	tonLimitPosMinReachedDelay	: TON;					// Timer osoiągniecia minimalnej wyskości 
	tonLimitPosMaxReachedDelay	: TON;					// Timer osiągnięcia maksymalnej wyskości
	tonSortingEngineOn			: TON;					// Opóźnienie po załączeniu napędu
	tonSortingEngineOff			: TON;					// Opóźnienie wyłączenia napędu
	tonSleeveFullEngineOn		: TON;					// Czas załączenia napędu po wykrciu braku nasadek
	tonEngineBlocked			: TON;					// Zablokowany silnik	
	rtCapSorterSensor			: R_TRIG;				// Triger
	tonTryUnblockWheel			: TON;					// Czas ruchu falownika w drugą stronę
	tofCapFeederSorterCapSensor	: TOF;					// Opóźnienie sygnału z czujnika obecności nasadki ultradzwiek
	tonCapFeederSorterCapSensor	: TON;					// Opóźnienie sygnału z czujnika obecności nasadki ultradźwięk
	tonAirBeforeStart			: TON;					// Czasówka opóźeniani przedmuchu
	tonAirBeforeStart2			: TON;					// Czasówka opóźeniani przedmuchu
	tonAirAfterStop				: TON;					// Czasówka przedmuchu po zatrzymaniu
	tonStoppingTime				: TON;					// Czasówka zbyt długiego zatrzymawania

	
	tonErrorHeightChange		: TON; 					// Timer błędu zacięcia się podnośnika
	tonMaxHeightError			: TON;					// Timer ustawienia zbyt dużej wysokości stacji
	tonMinHeightError			: TON;					// Timer ustawienia zbyt małej wysokości stacji
	tonCycleTimer				: TON;					// Czasówka cyklu
	rtrigCycleTimerRead			: R_TRIG;				// Trigger do statystyk cyklu 
	
	rtResetCommands				: R_TRIG;
	tonHomingSensor: TON;
	TimerOn: TON;
	TimerOff: TON;
	bImpOn: BOOL;
	rtCapFeederSorterCapSensor: R_TRIG;
	bBlowDelay: BOOL;
	tonbBlowDelay: TON;
	
	fbInverter: FB_MitsubishiInverter;
	fbInverter2: FB_MitsubishiInverter;	
	tonInverterError: TON;
	tonInverter2Error: TON;	
	tonbCapping1Tool2ActuatorUpError: TON;
	tonbCapping2Tool2ActuatorUpError: TON;	
	
	(*Ostrzeżenia*)
	fbbLevelSensor:	FB_InputFilter;
	(*Inne*)	

	tonGates1	:	TON;	//Czasówka dla szlabanów w rękawe
	tonGates2	:	TON;	//Czasówka dla szlabanów w rękawe
	tonGates3	:	TON;	//Czasówka dla szlabanów w rękawe
	tonGates4	:	TON;	//Czasówka dla szlabanów w rękawe

	toneHolding1 :TON;
	toneHolding2 :TON;
	toneGoingUp	:TON;
	toneHolding1Tool2 :TON;
	toneHolding2Tool2 :TON;
	
	bDone1				: BOOL;					// Sygnał o niezakończonym cyklu
	bDone2				: BOOL;					// Sygnał o niezakończonym cyklu
	
	tonDown1:TON;
	tonDown2:TON;	
	tonEnginesRun:TON;	
	tonDone	:TON;	
	ftbRunEngine: F_TRIG;
	bGates	    :	BOOL;	//Controla szłabanow w rękawe  
	bTryUnblockWheel : BOOL;
	iTryUnblockWheel : INT;
END_VAR

//Wywołanie bloczków od stacji. Ważna jest ich kolejność!!!
ACT_Limits();
ACT_HeightMotor();
ACT_ErrorHandling();

ACT_Signals();
ACT_Control();
aEngine();
ACT_Inverter();
ACT_Statistic();
ACT_Status();
ACT_Warnings();
aStationID();	

lrLastHeightMotorPositionCV:=lrHeightMotorCV;

ACTION ACT_Control:
	(*****Wyłączenie enable*****)
	IF NOT bEnable THEN
		IF eState <> E_Station.eDisabled AND eState <> E_Station.ePreparingToDisable THEN
				eState 				:= E_Station.ePreparingToDisable; 
		END_IF	
	END_IF

	(*****Estop*****)
	IF NOT bEstop  THEN	
		IF eState <> E_Station.eAborted AND eState <> E_Station.eAborting AND eState <> E_Station.eDisabled THEN
				eState 				:= E_Station.eAborting; 
		END_IF
	END_IF


	CASE eState OF
//--------------------------------------------------------------------------------
// Stan maszyny po wyłączeniu i przygotowanie do uruchomienia
	E_Station.eDisabled: 					// Stan nieaktywnosci (Stacja wyłączona) 
	
		IF bEnable THEN
			eState 				:= E_Station.ePreparingToReady; 
		END_IF 
		
//--------------------------------------------------------------------------------
// Stan maszyny po zatrzymaniu awaryjnym   
	E_Station.eAborted: 					// Stan bezpiecznego zatrzymania (po Abortingu) 

		IF bEStop THEN
			eState 				:= E_Station.ePreparingToReady;
		END_IF
		
//--------------------------------------------------------------------------------
// Stan maszyny naciśnieciu estopa 	
	E_Station.eAborting:                 	// Stan bezpiecznego zatrzymywania (po EStopie)

		ACT_ResetCommands();

		eState 						:=  E_Station.eAborted;  
		eRunningState				:=	E_GripperScrewer.eReady;
		
//--------------------------------------------------------------------------------
// Stan masyzny po wykryciu błędu			
	E_Station.eError:                 	 	// Stan błędu 	
		
		ACT_ResetCommands();
		
		IF bReset THEN
			eState 					:= E_Station.eResetting;
			bError					 := FALSE;
		END_IF
		
//--------------------------------------------------------------------------------
// Stan masyzny po wykryciu błędu
	E_Station.eResetting:					// Stan resetowania bledu (po Errorze)
			CASE udiErrorID OF
		
				//Error - Błąd falownika
				353,354:
					fbInverter.bReset	:= TRUE;
					fbInverter2.bReset	:= TRUE;					
					bError 				:= FALSE;
				ELSE
					bError := FALSE;	
			END_CASE		
		
		IF NOT bError AND fbInverter.eState = E_Station.eReady THEN
			fbInverter.bReset	:= FALSE;	
			fbInverter2.bReset	:= FALSE;
			//{warning 'Sprawdzić błąd falownika CapFeeder'}
			udiErrorID 			:=	0;
			sErrorDescription 	:=	'';
			eState 				:=	E_Station.ePreparingToReady;
			eRunningState		:=	E_GripperScrewer.eReady;
		ELSE
			eState 				:=	E_Station.eError;
		END_IF
    
//--------------------------------------------------------------------------------
// Stan ruchoow manualnych
	E_Station.eManualMovement:     			// Stan ruchów manualnych  
   
		ACT_ManualMovements();
		//Wyjście z trybu serwisowego
		IF NOT bManualMovement THEN
			bHeightMotorUp				:=	FALSE;
			bHeightMotorDown			:=	FALSE;
			eState:=E_Station.eReady;
		END_IF
		
//--------------------------------------------------------------------------------
// Stan rozpoczecia bazowania
	E_Station.eHoming:						// Stan bazowania 
		
		ACT_Homing();
		IF NOT bHoming AND NOT bHeightSet THEN
			bHeightMotorDown				:=	FALSE;
			bHeightMotorUp					:=	FALSE;
		   eState							:=	E_Station.ePreparingToReady;
		END_IF		
		
//--------------------------------------------------------------------------------
// Stan zakończenia bazowania
	E_Station.eHomingDone:                  // Stan wykonania bazowania 
	
		bHeightMotorDown					:=	FALSE;
		bHeightMotorUp						:=	FALSE;
		bHeightMotorEncoderCounterReset		:=	FALSE;
		bHomingDone							:=	TRUE;
		IF NOT bHoming AND NOT bHeightSet THEN
		   eState:=E_Station.eReady;
		END_IF
		
//--------------------------------------------------------------------------------
// Stan przygotowania do gotowości
	E_Station.ePreparingToReady:            // Stan przygotowywania do gotowosci (zawsze przed Ready)  

		eRunningState	:=	E_GripperScrewer.eReady;
		eState			:=	E_Station.eReady;	
		
//-------------------------------------------------------------------------------
// Stan przygotowania do wyłączenia maszyny
	E_Station.ePreparingToDisable:          // Stan przygotowywania do nieaktywnosci (po wyłączeniu Enable) 

		bHeightMotorUp		:=	TRUE;
		bHeightMotorDown	:=	FALSE;	
		IF tonHeightNoChange.Q OR tonHeightNoChangeTime.Q THEN
			bHeightMotorUp			:=	FALSE;
			bHeightMotorDown		:=	FALSE;	
			eRunningState			:=	E_GripperScrewer.eReady;		
			eState					:=	E_Station.eDisabled;
		END_IF	
			
//--------------------------------------------------------------------------------
// Stan gotowości
	E_Station.eReady:						// Stan gotowosci 
	
		(*Skasowanie wszystkich komend*)
		IF rtResetCommands.Q THEN	ACT_ResetCommands();	END_IF
	
		IF (bRun1 OR bRun2) AND NOT bCycleDone1 AND NOT bCycleNotDone1 AND NOT bCycleDone2 AND NOT bCycleNotDone2 THEN
			eState 				:= E_Station.eStarting; 
		END_IF
		IF bHoming OR bHeightSet THEN
			eState 				:= E_Station.eHoming; 
		END_IF
		IF bManualMovement THEN
			bManualHeightMotorUp					:=	bHeightMotorUp;					
			bManualHeightMotorDown				:=	bHeightMotorDown;	
			bManualEngine1						:=	fbInverter.bRun;							
			bManualEngine2						:=	fbInverter2.bRun;		
			bManualCapping1Tool1Actuator		:=	bCapping1Tool1Actuator;		
			bManualCapping2Tool1Actuator		:=	bCapping2Tool1Actuator;		
			bManualCapping12Tool1BlockActuator	:=	bCapping12Tool1BlockActuator;
			bManualCappingBlockActuator			:=	bCappingBlockActuator;	
			bManualCapping1Tool2Down			:=	bCapping1Tool2Down;	
			bManualCapping1Tool2Tight			:=	bCapping1Tool2Tight;			
			bManualCapping1Tool2Realese			:=	bCapping1Tool2Realese;		
			bManualCapping2Tool2Down			:=	bCapping2Tool2Down;				
			bManualCapping2Tool2Tight			:=	bCapping2Tool2Tight;
			bManualCapping2Tool2Realese			:=	bCapping2Tool2Realese;
			bManualFormPositioning				:=	bFormPositioning;			
			eState 								:=	E_Station.eManualMovement; 
		END_IF
		IF NOT bRun1 AND NOT bRun2 THEN
			bDone1						:= FALSE;
			bDone2						:= FALSE;
			bCycleDone1 				:= FALSE;
			bCycleNotDone1 				:= FALSE;	
			bCycleDone2					:= FALSE;
			bCycleNotDone2 				:= FALSE;	
			bWarning1					:= FALSE;	
		END_IF
		
//--------------------------------------------------------------------------------
// Stan zatrzymywania
	E_Station.eStopping:					// Stan zatrzymywania 
		
		ACT_Running();

		IF tonStoppingTime.Q THEN
			ACT_ResetCommands();
			eRunningState							:= E_GripperScrewer.eReady;
			eState									:= E_Station.eReady;
		END_IF

		
//--------------------------------------------------------------------------------
// Stan uruchomienia lini ( po eReady)
	E_Station.eStarting:                  	// Stan uruchamiania (po Ready)

		eState					 := E_Station.eRunning; 

//--------------------------------------------------------------------------------
// Stan wykonywania pracy
	E_Station.eRunning:               		// Stan wykonywania cyklu (po Startingu), w tym stanie osobny

		ACT_Running();
		IF NOT bRun1 AND NOT bRun2 THEN					(*Przerywanie cyklu*)
			eState 				 := E_Station.eStopping;	
		END_IF
		IF (bCycleDone1 OR bCycleNotDone1) AND (bCycleDone2 OR bCycleNotDone2)  THEN (*Cykl zakończony*)
			eState 				 := E_Station.eReady;
		END_IF						
		
		
END_CASE
END_ACTION

ACTION ACT_ErrorHandling:
//OBSŁUGA BŁĘDÓW STACJI SPRAWDZANIA
//************LISTA BŁĘDÓW***************
bStateError:= (eState=E_Station.eError) OR (eState=E_Station.eResetting) OR bIgnoreError;
//************LISTA BŁĘDÓW***************

//Error 1 - podnośnik nie porusza się pomimo wysterowania 
tonErrorHeightChange(IN:=(bHeightMotorUp OR bHeightMotorDown) AND lrLastHeightMotorPositionCV=lrHeightMotorCV, PT:=T#3S);
tonMaxHeightError	(IN:=lrHeightMotorSV>lrMaxHeight AND NOT bHomingNeeded AND eState=E_Station.eReady,PT:=T#30S);
tonMinHeightError	(IN:=lrHeightMotorSV<lrMinHeight AND NOT bHomingNeeded AND eState=E_Station.eReady,PT:=T#30S);
tonInverterError	(IN:=fbInverter.bError AND NOT bStateError, PT:=T#3S);
tonInverter2Error	(IN:=fbInverter2.bError AND NOT bStateError, PT:=T#3S);

tonbCapping1Tool2ActuatorUpError (IN:= iTool = 2 (*G.dociskająca*) AND NOT IbCapping1Tool2ActuatorUpSensor AND NOT bCapping1Tool2Down, PT:=T#2S);
tonbCapping2Tool2ActuatorUpError (IN:= iTool = 2 (*G.dociskająca*) AND NOT IbCapping2Tool2ActuatorUpSensor AND NOT bCapping2Tool2Down, PT:=T#2S);

IF (bEnable OR (eState = E_Station.ePreparingToDisable)) AND NOT bIgnoreError THEN
	
	IF tonErrorHeightChange.Q THEN
		bError:=TRUE;
		udiErrorID:=350;
		sErrorDescription:='Blokada podnośnika lub brak zasilania - sprawdź czujnik lub odblokuj mechanicznie';	
		sErrorDescription2:='';
	END_IF
	
	//Error - Bład nastaw max
	IF tonMaxHeightError.Q  THEN
		bError:=TRUE;
		udiErrorID:=351;
		sErrorDescription:='Wartość zadana wysokości jest większa od maksymalnej - zmień ustawienia w recepturze';
		sErrorDescription2:=REAL_TO_STRING(LREAL_TO_INT(lrMaxHeight));
	END_IF
	
	//Error - Bład nastaw min
	IF tonMinHeightError.Q THEN
		bError:=TRUE;
		udiErrorID:=352;
		sErrorDescription:='Wartość zadana wysokości jest mniejsza od minimalnej - zmień ustawienia w recepturze';
		sErrorDescription2:=REAL_TO_STRING(LREAL_TO_INT(lrMinHeight));
	END_IF	
	
	//Error - Bład falownika 1
	IF tonInverterError.Q THEN
		bError:=TRUE;
		udiErrorID:=353;
		sErrorDescription:='Błąd falownika głowicy 1';
		sErrorDescription2:='';
	END_IF		
	
	//Error - Bład falownika 2
	IF tonInverter2Error.Q THEN
		bError:=TRUE;
		udiErrorID:=354;
		sErrorDescription:='Błąd falownika głowicy 2';
		sErrorDescription2:='';
	END_IF			
	
	//Error Glowica 1 - Bład góry
	IF tonbCapping1Tool2ActuatorUpError.Q THEN
		bError:=TRUE;
		udiErrorID:=355;
		sErrorDescription:='Błąd górnej pozycji głowicy dociskającej 1- upewnij się że jest wybrane dobre narzędzie lub sprawdź czujnik';
		sErrorDescription2:='';	
	END_IF			
	//Error Glowica 2 - Bład góry
	IF tonbCapping2Tool2ActuatorUpError.Q THEN
		bError:=TRUE;
		udiErrorID:=356;
		sErrorDescription:='Błąd górnej pozycji głowicy dociskającej 2 - upewnij się że jest wybrane dobre narzędzie lub sprawdź czujnik';
		sErrorDescription2:='';	
	END_IF			
	
ELSE
	bError	:=FALSE;
END_IF


//-----------------------------------------------------------------------
IF bError AND NOT bStateError THEN

	IF eLastState = eRunning THEN
		bCycleNotDone1						:= TRUE;
	END_IF

	eState 									:= E_Station.eError;
END_IF


//------------------------------------------------------------------------

(*Wyświetlanie błedu na wyjściu*)
bError;

(*Przepisywanie nazwy stacji*)
sErrorStationName 							:= sStationName;

//Jezeli nie zbazowane to potrzebne bazowanie
IF NOT bHeightMotorEncoderHomed  THEN
	bHomingDone								:=	FALSE;
END_IF
END_ACTION

ACTION ACT_HeightMotor:
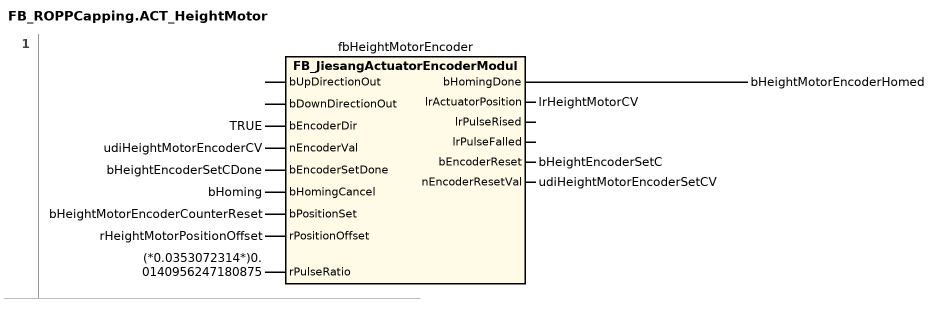
// NETWORK 1
fbHeightMotorEncoder(
    bEncoderDir := TRUE,
    nEncoderVal := udiHeightMotorEncoderCV,
    bEncoderSetDone := bHeightEncoderSetCDone,
    bHomingCancel := bHoming,
    bPositionSet := bHeightMotorEncoderCounterReset,
    rPositionOffset := rHeightMotorPositionOffset,
    rPulseRatio := (*0.0353072314*)0.0140956247180875,
    lrActuatorPosition => lrHeightMotorCV,
    bEncoderReset => bHeightEncoderSetC,
    nEncoderResetVal => udiHeightMotorEncoderSetCV); // FB_JiesangActuatorEncoderModul
bHeightMotorEncoderHomed := fbHeightMotorEncoder.bHomingDone;
END_ACTION

ACTION ACT_Homing:
//BAZOWANIE

tofHeightMotorDown(IN:=bHeightMotorDown, PT:=T#1S); //Zabezpieczenie przed zbyt szybkim przełączeniem pomiędzy Down a Up, bezpiecznieki sie palą
	
//Podnoszenie stacji do maksymalnej pozycji
IF NOT bHeightMotorEncoderHomed OR rtEncoderHomed.Q THEN
	bHeightMotorUp:=(*TRUE*) NOT tofHeightMotorDown.Q AND NOT tonHomingSensor.Q;
	bHeightMotorDown:=FALSE;
	IF tonHeightNoChange.Q OR tonHeightNoChangeTime.Q THEN
		bHeightMotorEncoderCounterReset:=TRUE;
		bHeightMotorUp:=FALSE;
    END_IF
	//Jesli enkoder zbazowany zakończ bazowanie	
	IF rtEncoderHomed.Q  THEN
		bHeightMotorUp:=FALSE;
		bHeightMotorDown:=FALSE;
		eState:=E_Station.eHomingDone;
	END_IF		
		
//Po podniesieniu stacji opuszczanie do ustalonej wysokości
ELSIF bHeightMotorEncoderHomed THEN
	bHeightMotorEncoderCounterReset:=FALSE;
	bHeightMotorUp:=lrHeightMotorCV<=lrHeightMotorSV;
	bHeightMotorDown:=lrHeightMotorCV>=lrHeightMotorSV;
	//Kiedy stacja osiągnie wysokość zadaną
	IF ABS(lrHeightMotorCV-lrHeightMotorSV)<0.5 OR tonLimitPosMaxReachedDelay.Q OR tonLimitPosMinReachedDelay.Q THEN
		bHeightMotorDown:=FALSE;
		bHeightMotorUp:=FALSE;
		eState:=E_Station.eHomingDone;
	END_IF			
END_IF
END_ACTION

ACTION ACT_Inverter:
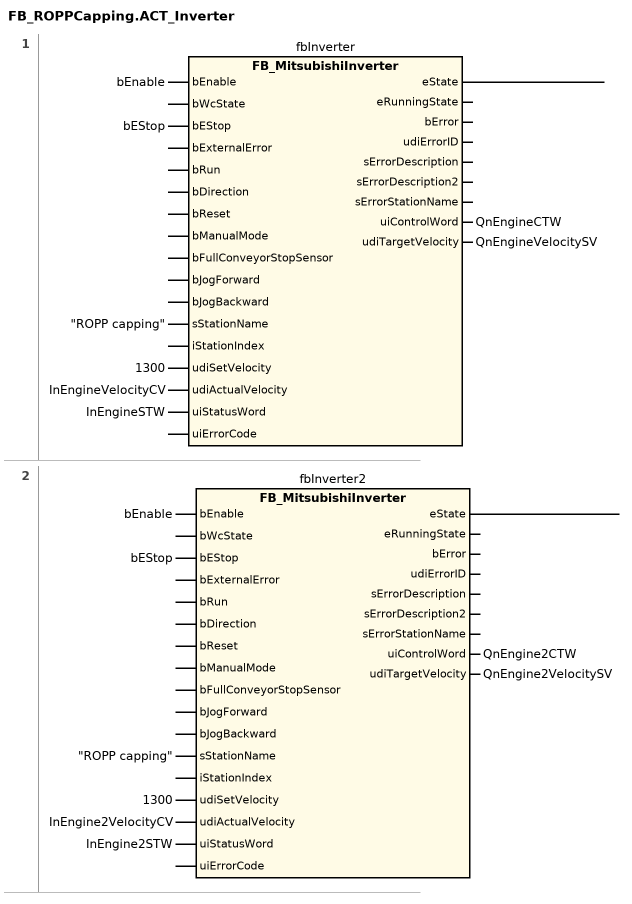
// NETWORK 1
fbInverter(
    bEnable := bEnable,
    bEStop := bEStop,
    sStationName := "ROPP capping",
    udiSetVelocity := 1300,
    udiActualVelocity := InEngineVelocityCV,
    uiStatusWord := InEngineSTW,
    uiControlWord => QnEngineCTW,
    udiTargetVelocity => QnEngineVelocitySV); // FB_MitsubishiInverter

// NETWORK 2
fbInverter2(
    bEnable := bEnable,
    bEStop := bEStop,
    sStationName := "ROPP capping",
    udiSetVelocity := 1300,
    udiActualVelocity := InEngine2VelocityCV,
    uiStatusWord := InEngine2STW,
    uiControlWord => QnEngine2CTW,
    udiTargetVelocity => QnEngine2VelocitySV); // FB_MitsubishiInverter
END_ACTION

ACTION ACT_Limits:

END_ACTION

ACTION ACT_ManualMovements:
//W trybie ruchów manualnych wykonuj ruchy za pomocą rozkazów manualnych
IF NOT bRun1 AND NOT bRun2 THEN
	
	bHeightMotorUp					:=	bManualHeightMotorUp;				
	bHeightMotorDown				:=	bManualHeightMotorDown;				
	fbInverter.bRun					:=	bManualEngine1;						
	fbInverter2.bRun				:=	bManualEngine2;						
	bCapping1Tool1Actuator			:=	bManualCapping1Tool1Actuator;		
	bCapping2Tool1Actuator			:=	bManualCapping2Tool1Actuator;		
	bCapping12Tool1BlockActuator	:=	bManualCapping12Tool1BlockActuator OR bManualCapping1Tool1Actuator OR bManualCapping2Tool1Actuator;	
	bCappingBlockActuator			:=	bManualCappingBlockActuator ;//OR bManualCapping1Tool1Actuator OR bManualCapping2Tool1Actuator;			
	bCapping1Tool2Down				:=	bManualCapping1Tool2Down;			
	bCapping1Tool2Tight				:=	bManualCapping1Tool2Tight;			
	bCapping1Tool2Realese			:=	bManualCapping1Tool2Realese;			
	bCapping2Tool2Down				:=	bManualCapping2Tool2Down;			
	bCapping2Tool2Tight				:=	bManualCapping2Tool2Tight;			
	bCapping2Tool2Realese			:=	bManualCapping2Tool2Realese;			
	bFormPositioning				:=	bManualFormPositioning;				

ELSE	//Kasuje zeby po cyklu nic sie nie poruszało

	bManualHeightMotorUp				:= FALSE;		
	bManualHeightMotorDown				:= FALSE;		
	bManualEngine1						:= FALSE;	
	bManualEngine2						:= FALSE;	
	bManualCapping1Tool1Actuator		:= FALSE;	
	bManualCapping2Tool1Actuator		:= FALSE;	
	bManualCapping12Tool1BlockActuator	:= FALSE;	
	bManualCappingBlockActuator			:= FALSE;	
	bManualCapping1Tool2Down			:= FALSE;	
	bManualCapping1Tool2Tight			:= FALSE;	
	bManualCapping1Tool2Realese			:= FALSE;	
	bManualCapping2Tool2Down			:= FALSE;	
	bManualCapping2Tool2Tight			:= FALSE;	
	bManualCapping2Tool2Realese			:= FALSE;	
	bManualFormPositioning				:= FALSE;	

END_IF

IF bHoming OR bHeightSet THEN
	eState:=E_Station.eHoming;
END_IF

IF bRun1 OR bRun2 THEN	
	ACT_Running();
END_IF

IF NOT bRun1 AND NOT bRun2 THEN
	bCycleDone1 				:= FALSE;
	bCycleNotDone1 				:= FALSE;	
	bCycleDone2					:= FALSE;
	bCycleNotDone2 				:= FALSE;	
	bWarning1					:= FALSE;	
END_IF

//Zabezpieczenie przed kolizją stacji poprzez ruch podnośnika	
IF bHeightMotorDown AND lrHeightMotorCV<=lrMinHeight AND NOT bHoming AND NOT bHeightSet THEN
	bHeightMotorDown:=FALSE;
END_IF	

IF bHeightMotorUp AND lrHeightMotorCV>=lrMaxHeight AND NOT bHoming AND NOT bHeightSet THEN
	bHeightMotorUp:=FALSE;
END_IF
END_ACTION

ACTION ACT_ResetCommands:
//Reset komend ruchu 	

bHeightMotorUp					:=	FALSE;
bHeightMotorDown				:=	FALSE;
fbInverter.bRun					:=	FALSE;
fbInverter2.bRun				:=	FALSE;
bCapping1Tool1Actuator			:=	FALSE;
bCapping2Tool1Actuator			:=	FALSE;
bCapping12Tool1BlockActuator	:=	FALSE;
bCappingBlockActuator			:=	FALSE;
bCapping1Tool2Down				:=	FALSE;
bCapping1Tool2Tight				:=	FALSE;
bCapping1Tool2Realese			:=	FALSE;
bCapping2Tool2Down				:=	FALSE;
bCapping2Tool2Tight				:=	FALSE;
bCapping2Tool2Realese			:=	FALSE;
bFormPositioning				:=	FALSE;
END_ACTION

ACTION ACT_Running:

CASE eRunningState OF

//====================================
	
	(*Oczekiwanie na wykonanie pojedynczego cyklu*)
	E_GripperScrewer.eReady:
	 		                                       	
		IF NOT bCycleDone1 AND NOT bCycleNotDone1 AND NOT bCycleDone2 AND NOT bCycleNotDone2 THEN                                           	
			IF bRun1 OR bRun2 THEN                			
					eRunningState						:=	E_GripperScrewer.eToPushingPosition;	
			END_IF
		END_IF
		
//====================================		
	(*Ruch na pozycję *)			
	E_GripperScrewer.eToPushingPosition:
	
		bFormPositioning				:= TRUE;
	
		bCapping12Tool1BlockActuator	:= TRUE;
		bCappingBlockActuator			:= TRUE;	
		
		IF		iTOOL = 1 THEN //Glowica zakręcająca
			fbInverter.bRun				:= bRun1;
			fbInverter2.bRun			:= bRun2;	

			IF bManualMode AND tonEnginesRun.Q THEN
				bCapping1Tool1Actuator		:= bRun1;
				bCapping2Tool1Actuator		:= bRun2;	
				eRunningState				:=	E_GripperScrewer.eScrewing;	
			ELSIF NOT bManualMode THEN
				bCapping1Tool1Actuator		:= bRun1;
				bCapping2Tool1Actuator		:= bRun2;	
				eRunningState				:=	E_GripperScrewer.eScrewing;	
			END_IF
			
		ELSIF	iTOOL = 2 THEN //Glowica dociskająca
			bCapping1Tool2Down			:= bRun1;	
			bCapping1Tool2Tight			:= FALSE;
			bCapping2Tool2Down			:= bRun2;
			bCapping2Tool2Tight			:= FALSE;
			eRunningState				:=	E_GripperScrewer.eScrewing;	
		END_IF
	

//====================================		
		
	(*Zakręcanie*)
	E_GripperScrewer.eScrewing:
	
		IF		iTOOL = 1 THEN //Glowica zakręcająca
			eRunningState					:=	E_GripperScrewer.eHolding;	
			
		ELSIF	iTOOL = 2 THEN //Glowica dociskająca
			
			IF tonDown1.Q THEN
				bCapping1Tool2Down			:=	bRun1;	
				bCapping1Tool2Tight			:=	bRun1;
				bCapping2Tool2Down			:=	bRun2;
				bCapping2Tool2Tight			:=	bRun2;
				eRunningState				:=	E_GripperScrewer.eHolding;
			END_IF
			
		END_IF	
	
//====================================

	(*Przytrzymanie / Czas na odbpuszczenie chwytakow*)					
	E_GripperScrewer.eHolding:
	
	
		IF		iTOOL = 1 THEN //Glowica zakręcająca
			IF (toneHolding1.Q OR NOT bRun1) THEN
				bDone1					:=	TRUE;
				bCapping1Tool1Actuator	:=	FALSE;
			END_IF
			IF (toneHolding2.Q OR NOT bRun2) THEN
				bDone2					:=	TRUE;				
				bCapping2Tool1Actuator	:=	FALSE;	
			END_IF	
			IF NOT 	bCapping1Tool1Actuator	AND NOT bCapping2Tool1Actuator THEN
				eRunningState					:=	E_GripperScrewer.eGoingUp;	
			END_IF
		ELSIF	iTOOL = 2 THEN //Glowica dociskająca

			IF (toneHolding1Tool2.Q OR IbCapping1Tool2ActuatorCappingDoneSensor OR NOT bRun1) THEN	
				bDone1						:=	IbCapping1Tool2ActuatorCappingDoneSensor;
				bCapping1Tool2Tight			:=	FALSE;
			END_IF
			
			IF (toneHolding2Tool2.Q OR IbCapping2Tool2ActuatorCappingDoneSensor OR NOT bRun2) THEN
				bDone2						:=	IbCapping2Tool2ActuatorCappingDoneSensor;		
				bCapping2Tool2Tight			:=	FALSE;
			END_IF	
			
			IF NOT 	bCapping1Tool2Tight	AND NOT bCapping2Tool2Tight THEN
				eRunningState				:=	E_GripperScrewer.eGoingUp;	
			END_IF			
	
		END_IF	

//====================================	

	(*Podnoszenie do góry / reset laga i obrót do pozycji gotowości*)			 
	E_GripperScrewer.eGoingUp:
	

		IF		iTOOL = 1 THEN //Glowica zakręcająca
			

			bCapping1Tool1Actuator			:=	FALSE;
			bCapping2Tool1Actuator			:=	FALSE;	
			bFormPositioning				:=	FALSE;			

			IF bManualMode THEN
				IF tonDone.Q THEN
					bCapping12Tool1BlockActuator	:= FALSE;
					bCappingBlockActuator			:= FALSE;
					fbInverter.bRun					:= FALSE;
					fbInverter2.bRun				:= FALSE;	
					eRunningState 					:=	E_GripperScrewer.eDone;					
				END_IF	
			ELSIF NOT bManualMode THEN	
					IF NOT bRunEngine THEN
						fbInverter.bRun					:= FALSE;
						fbInverter2.bRun				:= FALSE;	
						bCappingBlockActuator			:= FALSE;					
						eRunningState 					:=	E_GripperScrewer.eDone;	
					ELSE
						eRunningState 					:=	E_GripperScrewer.eDone;	
					END_IF			
			END_IF
		
		
		ELSIF	iTOOL = 2 THEN //Glowica dociskająca
			bCapping1Tool2Tight			:=	FALSE;		
			bCapping2Tool2Tight			:=	FALSE;	
	
			IF toneGoingUp.Q THEN
				bCapping1Tool2Down			:=	FALSE;		
				bCapping2Tool2Down			:=	FALSE;	
				eRunningState				:=	E_GripperScrewer.eDone;	
			END_IF
	
		END_IF	
		

		
//====================================			
	(*Zakręcono*)			
	E_GripperScrewer.eDone:
	
		bCycleDone1 						:=	bRun1 AND bDone1;
		bCycleNotDone1						:=	NOT bRun1 OR NOT bDone1;
		bCycleDone2 						:=	bRun2 AND bDone2;
		bCycleNotDone2						:=	NOT bRun2 OR NOT bDone2;	
	
		eRunningState 					:=	E_GripperScrewer.eReady;					


//====================================	
			
	E_GripperScrewer.eNotDone:

		bCycleNotDone1 						:=	TRUE;
		bCycleNotDone2						:=	TRUE;
		eRunningState						:=	E_GripperScrewer.eReady;	
	
END_CASE
END_ACTION

ACTION ACT_Signals:
(** Timery na potrzeby bazowania**)
rtEncoderHomed(CLK:=bHeightMotorEncoderHomed,Q=>);
tonHeightNoChange(IN:=((bHeightMotorUp OR bHeightMotorDown OR tonHomingSensor.Q) AND (lrLastHeightMotorPositionCV=lrHeightMotorCV)), PT:=T#500MS); 


tonLimitPosMinReachedDelay(IN:=(lrHeightMotorCV<=lrMinHeight) AND eState=E_Station.eHoming,PT:=T#2S);
tonLimitPosMaxReachedDelay(IN:=(lrHeightMotorCV>=lrMaxHeight) AND eState=E_Station.eHoming,PT:=T#2S);

rtResetCommands			(CLK:=	eState = E_Station.eReady (* OR *)		,Q=>); //Triger do resetu zmienych


(** Timery używane podczas pracy stacji**)
toneHolding1	(IN:=	eRunningState=E_GripperScrewer.eHolding AND IbCapping1Tool1ActuatorDownSensor, PT:= INT_TO_TIME(iTime));
toneHolding2	(IN:=	eRunningState=E_GripperScrewer.eHolding AND IbCapping2Tool1ActuatorDownSensor, PT:= INT_TO_TIME(iTime));	

toneHolding1Tool2	(IN:=	eRunningState=E_GripperScrewer.eHolding AND bCapping1Tool2Down, PT:= INT_TO_TIME(2000));
toneHolding2Tool2	(IN:=	eRunningState=E_GripperScrewer.eHolding AND bCapping2Tool2Down, PT:= INT_TO_TIME(2000));	

toneGoingUp			(IN:=	eRunningState=E_GripperScrewer.eGoingUp , PT:= T#300MS);	


tonDown1		(IN:=	eRunningState=E_GripperScrewer.eScrewing, PT:= INT_TO_TIME(iTime2));
tonDown2		(IN:=	eRunningState=E_GripperScrewer.eScrewing, PT:= INT_TO_TIME(iTime2));	

tonEnginesRun	(IN:= fbInverter.bRun OR fbInverter2.bRun, PT:=T#1S);
tonDone			(IN:= eRunningState = E_GripperScrewer.eGoingUp, PT:=T#1S);

ftbRunEngine	(CLK:=bRunEngine,Q=>);

(** Dodatkowy timer przy zatrzymywaniu**)
tonStoppingTime( IN:= eState= E_Station.eStopping, PT:=T#2S);
END_ACTION

ACTION ACT_Statistic:
//Statystyka do zliczania czasu cyklu 
rtrigCycleTimerRead(CLK:=eRunningState=E_GripperScrewer.eDone );

	IF rtrigCycleTimerRead.Q THEN
		tCycleTime:=tonCycleTimer.ET;
		
	END_IF
	
	tonCycleTimer(IN:=eRunningState>E_GripperScrewer.eReady,PT:=T#1D);
END_ACTION

ACTION ACT_Status:

(*Zapisywanie ostatniego stanu*)
	IF eLastStateTemp<>eState THEN
		eLastState := eLastStateTemp;
	END_IF
	eLastStateTemp := eState;
	
	IF eLastRunningStateTemp<>eRunningState THEN
		eLastRunningState := eLastRunningStateTemp;
	END_IF
	eLastRunningStateTemp := eRunningState;
(*Koniec Zapisywanie ostatniego stanu*)
END_ACTION

ACTION ACT_Warnings:

END_ACTION

ACTION aEngine:

IF bRunEngine THEN
	fbInverter.bRun				:=	TRUE;	
	fbInverter2.bRun			:=	TRUE;		
	bCappingBlockActuator		:=	TRUE;
END_IF

IF ftbRunEngine.Q THEN
	fbInverter.bRun				:=	FALSE;	
	fbInverter2.bRun			:=	FALSE;		
	bCappingBlockActuator		:=	FALSE;
END_IF
END_ACTION

ACTION aStationID:
udiStationID	:=	udiStationIndex;
END_ACTION

END_FUNCTION_BLOCK

// ---- POUs/FB/FB_IfmIoLinkRfid.TcPOU
//-----------------------------------------------------------------------------------------------------
//																
//									 	Tkmatik sp. z o.o.
//
//	Name				:		FB_IfmIoLinkRfid
//  Author				:		AM
//	Release Date		:		06.07.2022
//  Current ver			:		v 0.1
// 	Last correction 	:		06.07.2022
// 
//	Description			:						
//	This functional block operate with IFM RFID reader (for example DTI515), connected to PLC via IOLink
//	Allow user to read USER data from RFID tags.
//	1) bReadEnable = true enable asyncronious RFID reading. When DATA is readed FB set bCodeReaded until
//	tag is in reading zone, readed code saved into aReadCode. 
//	bCodeReaded set true if readed code <> last readed code
//	2) For writ USER data to tag: set new code into aWriteCode, than set bWriteEnable = true
//	When system set bWriteDone, code has been writed into tag, bWriteDone resets when bWriteEnable = false
//	4) aIoLinkInputData, bIoLinkTagPresent, nIoLinkErrorValue, bIoLinkCmdEnd, nIoLinkDataCounterIn,
//  bIoLinkCmdStartAck must be connected to IOLink IN; bIoLinkCmdStart, nIoLinkCmmandValue, nIoLinkDataCounter
//	nIoLinkDataCounter must be connecter do IOLink OUT
//
//	Requared hardware	:
//	IFM DTE515 (or other IFM), connected to IOLink
//
//-----------------------------------------------------------------------------------------------------

FUNCTION_BLOCK FB_IfmIoLinkRfid
VAR_INPUT
	//Commands
	bReadEnable						:		BOOL;					//Enable reading USER tag -> aReadCode
	bWriteCmd						:		BOOL;					//Command write aWriteData -> USER tag 
	//Data
	diWriteData						:		DINT;

	//IOLink connection
	aIoLinkInputData  			: 		ARRAY[0..27] OF USINT;
	bIoLinkTagPresent			:		BOOL;
	nIoLinkErrorValue			:		BYTE;
	bIoLinkCmdEnd				:		BOOL;
	nIoLinkDataCounterIn		:		BYTE;
	bIoLinkCmdStartAck			:		BOOL;
	
	
END_VAR

VAR_OUTPUT
	//States and out data
	bCodeReaded						:		BOOL;					//Flag tag on reader 
	bNewCodeReaded					:		BOOL;					//Flag NEW tag on reader
	bWriteCycleEnd					:		BOOL;					//Flag write operation done
	bBysy							:		BOOL;					//Reading or writing operation in process
	diReadedCode					:		DINT;
	bError							:		BOOL;					//RFID sensor error			
	sErrorDescription				:		STRING;					//Error description via Manual
	
	//IOLink connection
	bIoLinkCmdStart				:		BOOL;
	nIoLinkCmmandValue			:		BYTE;
	nIoLinkDataCounterOut		:		BYTE;
	aIoLinkOutputData  			: 		ARRAY[0..27] OF USINT;
END_VAR

VAR
	fbDIntTo4Byte					:		FB_DIntTo4Byte;
	aWriteData						:		ARRAY[0..15] OF BYTE;	//User data for writing	
	nWriteLengthLo					:		BYTE:=4;					//Length ou user data (max = 16)
	
	aReadCode						:		ARRAY [0..15] OF BYTE;	//Readed code value (saved)

	
	i								:		INT;					//FOR iterator
	
	//Read variables
	aReadCodeOld					:		ARRAY [0..15] OF BYTE;	//Readed code value (saved)
	rtReadFlag						:		R_TRIG;					//Tag on sensor trig
	iRead							:		INT;					//Read cycle case
	
	//Write variables
	iWrite							:		INT;					//Write cycle case
	rtWriteCmd						:		R_TRIG;					//New write command
	ftWriteCmd						:		F_TRIG;					//Write command off (for reset DONE signal)
END_VAR

VAR CONSTANT
	//Config
	nRegUserTagAdressHi				:		INT		:= 2;			//See user's manual
	nRegUserTagAdressLo				:		INT		:= 3;		    //See user's manual
	nRegUserTagLengthHi				:		INT		:= 4;			//See user's manual
	nRegUserTagLengthLo				:		INT		:= 5;		    //See user's manual
	nWriteLengthHi					:		BYTE	:= 0;			//We use only first 16 byte of tag

	//Operations
	nNoOperationCommand				:		BYTE	:= 16#04;		//Value of command register NOP
	nWriteUserDataCommand			:		BYTE	:= 16#04;		//Value of command register WR
	nReadUserDataCommand			:		BYTE	:= 16#01;		//Value of command register RD
	nBaseUserTagAdreessHi			:		BYTE	:= 16#00;		//Defaul adress of User data, we use only max first 16 byte;
	nBaseUserTagAdreessLo			:		BYTE	:= 16#00;		//Defaul adress of User data, we use only max first 16 byte;
END_VAR

aErrorHandling();
aMain();

ACTION aErrorHandling:
bError		 							:= nIoLinkErrorValue >0;

CASE nIoLinkErrorValue OF

	16#00	:	sErrorDescription		:= '';
	16#01	:	sErrorDescription		:= 'RFID UNKNOWN COMMAND';
	16#11	:	sErrorDescription		:= 'COMMAND NO RESPONSE';
	16#12	:	sErrorDescription		:= 'COMMAND RX ERROR';
	16#21	:	sErrorDescription		:= 'TAG COMMAND NOT SPECIFIED';
	16#22	:	sErrorDescription		:= 'TAG COMMAND SYNTAX';
	16#23	:	sErrorDescription		:= 'TAG OPTION NOT SUPPORTED';
	16#2F	:	sErrorDescription		:= 'TAG OTHER ERROR';
	16#30	:	sErrorDescription		:= 'TAG BLOCK NOT USABLE';
	16#31	:	sErrorDescription		:= 'TAG BLOCK ALREADY BLOCKED';
	16#32	:	sErrorDescription		:= 'TAG BLOCK NOT UPDATEBLE';
	16#33	:	sErrorDescription		:= 'TAG BLOCK WRITE VERIFY';
	16#34	:	sErrorDescription		:= 'TAG BLOCK LOCK VERIFY';
	ELSE
		sErrorDescription				:= 
			CONCAT(STR1 				:= 'UNKNOWN ERROR CODE = 0x',
				   STR2 				:= BYTE_TO_HEXSTR(in:=nIoLinkErrorValue,iPrecision:=2,bLoCase:=TRUE));
END_CASE
END_ACTION

ACTION aMain:
IF (iRead = 0 AND iWrite = 0) THEN
	bIoLinkCmdStart						:= FALSE;
	nIoLinkCmmandValue					:= nNoOperationCommand;
END_IF

//Read operations
IF (bReadEnable AND iWrite = 0 AND iRead = 0) THEN
	iRead								:= 1;
END_IF

//Write operation
rtWriteCmd(CLK:=bWriteCmd);
ftWriteCmd(CLK:=bWriteCmd);
IF (rtWriteCmd.Q AND iWrite = 0 AND iRead=0) THEN
	iWrite								:= 1;
END_IF
IF ftWriteCmd.Q THEN
	bWriteCycleEnd						:= FALSE;
	iWrite 								:= 0;
END_IF

//Actions calling
aWrite();
aRead();

bBysy									:=	iRead > 0 OR iWrite > 0;
END_ACTION

ACTION aRead:
CASE iRead OF
	0:
		;
	1:
		bIoLinkCmdStart					:= FALSE;
		iRead							:= 2;
	2:
		nIoLinkCmmandValue	 			:= nReadUserDataCommand; // read user data
		bIoLinkCmdStart					:= TRUE;
		iRead							:= 3;
	3:
		rtReadFlag(CLK := (bIoLinkTagPresent AND bIoLinkCmdEnd));
		
		IF (rtReadFlag.Q) THEN
			FOR i:=0 TO 15 DO
		
				IF (aReadCode[i] <> USINT_TO_BYTE( aIoLinkInputData[i])) THEN
					bNewCodeReaded		:= TRUE;
				END_IF
		
				aReadCode[i] 			:= USINT_TO_BYTE( aIoLinkInputData[i]);
		
			END_FOR
			diReadedCode				:=	DWORD_TO_DINT(F_4BYTES_TO_DWORD(BByte0:=aReadCode[3],BByte1:=aReadCode[2],BByte2:=aReadCode[1],BByte3:=aReadCode[0]));
				
			//iReadedCode					:= F_2Bytes_To_Word(byHigh:=aReadCode[4],byLow:=aReadCode[3]); 
		END_IF

		bCodeReaded  							:= bIoLinkTagPresent AND bIoLinkCmdEnd;

		IF (NOT bCodeReaded) THEN
			bNewCodeReaded						:= FALSE;
		END_IF
		
		IF (NOT bReadEnable) THEN
			FOR i:=0 TO 15 DO
				aReadCodeOld[i]					:= 0;
			END_FOR
			bCodeReaded							:= FALSE;
			bNewCodeReaded						:= FALSE;
			iRead								:= 0;
		END_IF
END_CASE
END_ACTION

ACTION aWrite:
CASE iWrite OF
	0:
		;
	1:
		IF (bIoLinkTagPresent) THEN
			iWrite								:= 2;
		END_IF
	2:
		bIoLinkCmdStart							:= FALSE;
		iWrite									:= 3;
	3:
		nIoLinkCmmandValue	 					:= nWriteUserDataCommand;
		
		aIoLinkOutputData[0]					:= 0;
		aIoLinkOutputData[1]					:= 0;
		
		aIoLinkOutputData[nRegUserTagAdressHi]	:= nBaseUserTagAdreessHi;
		aIoLinkOutputData[nRegUserTagAdressLo]	:= nBaseUserTagAdreessLo;
		aIoLinkOutputData[nRegUserTagLengthHi]	:= nWriteLengthHi;
		aIoLinkOutputData[nRegUserTagLengthLo]	:= nWriteLengthLo;
		
		aIoLinkOutputData[6]					:= 0;
		aIoLinkOutputData[7]					:= 0;
		aIoLinkOutputData[8]					:= 0;
		aIoLinkOutputData[9]					:= 0;
		aIoLinkOutputData[10]					:= 0;
		aIoLinkOutputData[11]					:= 0;
		aIoLinkOutputData[12]					:= 0;
		aIoLinkOutputData[13]					:= 0;
		aIoLinkOutputData[14]					:= 0;
		aIoLinkOutputData[15]					:= 0;
		aIoLinkOutputData[16]					:= 0;
		aIoLinkOutputData[17]					:= 0;
		aIoLinkOutputData[18]					:= 0;
		aIoLinkOutputData[19]					:= 0;
		aIoLinkOutputData[20]					:= 0;
		aIoLinkOutputData[21]					:= 0;
		aIoLinkOutputData[22]					:= 0;
		aIoLinkOutputData[23]					:= 0;
		aIoLinkOutputData[24]					:= 0;
		aIoLinkOutputData[25]					:= 0;
		aIoLinkOutputData[26]					:= 0;

		nIoLinkDataCounterOut					:= 0;
		bIoLinkCmdStart							:= TRUE;
		iWrite									:= 4;
	4:
		IF (bIoLinkCmdStartAck) THEN
			iWrite								:= 5;
		END_IF
	5:
		fbDIntTo4Byte(iInput:=diWriteData,by0=>aWriteData[0],by1=>aWriteData[1],by2=>aWriteData[2],by3=>aWriteData[3]);

		FOR i:=0 TO (nWriteLengthLo-1) DO
			aIoLinkOutputData[i]				:= aWriteData[i];
		END_FOR
		FOR i:=nWriteLengthLo TO 26 DO
			aIoLinkOutputData[i]				:= 0;
		END_FOR
		nIoLinkDataCounterOut					:= 1;
		iWrite									:= 6;
	6:
		IF (nIoLinkDataCounterIn = 1) THEN
			iWrite								:= 7;
		END_IF
	7:
		IF (bIoLinkCmdEnd) THEN
			iWrite									:= 0;	
			bWriteCycleEnd							:= TRUE;
		END_IF	
END_CASE
END_ACTION

END_FUNCTION_BLOCK

// ---- POUs/FB/Conversions/FB_DIntTo4Byte.TcPOU
(****************************************************************************************)
(*							Beckhoff Automation Poland									*)
(*								FB_IntTo2Byte	 v1.0									*)
(*									24.5.2011											*)
(*			Blok funkcyjny rozbijający zmienną typu INT na dwie zmienne typu BYTE		*)
(*______________________________________________________________________________________*)
FUNCTION_BLOCK FB_DIntTo4Byte
VAR_INPUT
	iInput :DINT;
END_VAR
VAR_OUTPUT
	by0 : BYTE;
	by1 : BYTE;
	by2 : BYTE;
	by3 : BYTE;
END_VAR

by3 := DINT_TO_BYTE(iInput);
by2 := DINT_TO_BYTE(SHR(iInput, 8));
by1 := DINT_TO_BYTE(SHR(iInput, 16));
by0 := DINT_TO_BYTE(SHR(iInput, 24));

END_FUNCTION_BLOCK

// ---- POUs/FB/Conversions/F_4BYTES_TO_DWORD.TcPOU
(****************************************************************************)
(*							Beckhoff Automation Poland						*)
(*							F_4BYTES_TO_DWORD v1							*)
(*									21.11.2013								*)
(*					Funkcja zamieniająca 4 zmienne typu BYTE na DWORD 		*)
(*__________________________________________________________________________*)
FUNCTION F_4BYTES_TO_DWORD : DWORD
VAR_INPUT
	BByte0		: BYTE;
	BByte1		: BYTE;
	BByte2		: BYTE;
	BByte3		: BYTE;
END_VAR

F_4BYTES_TO_DWORD := BByte3 *16#1000000 + BByte2 *16#10000 + BByte1 *16#100 + BByte0;

END_FUNCTION

// ---- POUs/P15_FormTransporters.TcPOU
(*
Nazwa:			P15_FormTransporters
Opis:			Stacja transporterow
Wersja:			v0.1
Data:			2025-06-02
Autor:			DP
Urzadzenia:		
Konfiguracja:	
Info:

*)

PROGRAM P15_FormTransporters
VAR

	(*****************TRANSPORTER BUTELEK*******************)
	fbFormTransporterDispencer								: FB_MitsubishiInverter;
	eFormTransporterDispencerState							: E_Station;			
	eFormTransporterDispencerRunningState					: E_ConveyorState;	
	fbFormTransporterDispencerState							: FB_State;		
	QnFormTransporterDispencerVelocitySV					AT %Q*: UDINT; 			(*po kom*)	// Nastawa prędkości transportera
	InFormTransporterDispencerVelocityCV 					AT %I*: UDINT;			(*po kom*)
	InFormTransporterDispencerSTW 							AT %I*: UINT; 			(*po kom*)	// Statusword transportera wejściowego
	QnFormTransporterDispencerCTW 							AT %Q*: UINT;  			(*po kom*)	// Controlword transportera wejsciowego
	InFormTransporterDispencerErrorCode 					AT %I*: UINT;			(*po kom*)

	(*****************TRANSPORTER Za DOZOWNIKAMI******************)
	fbFormTransporterScrewer								 : FB_MitsubishiInverter;
	eFormTransporterScrewerState							 : E_Station;			
	eFormTransporterScrewerRunningState						 : E_ConveyorState;	
	fbFormTransporterScrewerState							 : FB_State;		
	QnFormTransporterScrewerVelocitySV 				  		 AT %Q*: UDINT; 		(*po kom*)	// Nastawa prędkości transportera
	InFormTransporterScrewerVelocityCV 						 AT %I*: UDINT;			(*po kom*)
	InFormTransporterScrewerSTW 							 AT %I*: UINT; 			(*po kom*)	// Statusword transportera wyjściowego
	QnFormTransporterScrewerCTW 							 AT %Q*: UINT;  		(*po kom*)	// Controlword transportera wyjsciowego
	InFormTransporterScrewerErrorCode						 AT %I*:UINT;			(*po kom*)
	
		(*****************TRANSPORTER PRZED ROPP*******************)
	fbFormTransporterROPP											 : FB_MitsubishiInverter;
	eFormTransporterROPPState										 : E_Station;			
	eFormTransporterROPPRunningState								 : E_ConveyorState;	
	fbFormTransporterROPPState										 : FB_State;		
	QnFormTransporterROPPVelocitySV 				  				 AT %Q*: UDINT; 		(*po kom*)	// Nastawa prędkości transportera
	InFormTransporterROPPVelocityCV 								 AT %I*: UDINT;			(*po kom*)
	InFormTransporterROPPSTW 										 AT %I*: UINT; 			(*po kom*)	// Statusword transportera wyjściowego
	QnFormTransporterROPPCTW 										 AT %Q*: UINT;  		(*po kom*)	// Controlword transportera wyjsciowego
	InFormTransporterROPPErrorCode									 AT %I*:UINT;			(*po kom*)
	
	(*****************TRANSPORTER  ZA SORTEREM NASADEK*******************)
	fbFormTransporterAfterCapSorter									: FB_MitsubishiInverter;
	eFormTransporterAfterCapSorterState								: E_Station;			
	eFormTransporterAfterCapSorterRunningState						: E_ConveyorState;	
	fbFormTransporterAfterCapSorterState							: FB_State;		
	QnFormTransporterAfterCapSorterVelocitySV 						AT %Q*: UDINT; 					// Nastawa prędkości transportera
	InFormTransporterAfterCapSorterVelocityCV 						AT %I*: UDINT;					
	InFormTransporterAfterCapSorterSTW 								AT %I*: UINT; 					// Statusword transportera wyjściowego
	QnFormTransporterAfterCapSorterCTW 								AT %Q*: UINT;  					// Controlword transportera wyjsciowego
	InFormTransporterAfterCapSorterErrorCode 						AT %I*: UINT;					
	
	(*****************TRANSPORTER PRZED ZAKRECARKAMI*******************)
	fbFormTransporterBeforeScrewer									: FB_MitsubishiInverter;
	eFormTransporterBeforeScrewerState								: E_Station;			
	eFormTransporterBeforeScrewerRunningState						: E_ConveyorState;	
	fbFormTransporterBeforeScrewerState								: FB_State;		
	QnFormTransporterBeforeScrewerVelocitySV 						AT %Q*: UDINT; 			(*po kom*)	// Nastawa prędkości transportera
	InFormTransporterBeforeScrewerVelocityCV 						AT %I*: UDINT;			(*po kom*)
	InFormTransporterBeforeScrewerSTW 								AT %I*: UINT; 			(*po kom*)	// Statusword transportera wyjściowego
	QnFormTransporterBeforeScrewerCTW 								AT %Q*: UINT;  			(*po kom*)	// Controlword transportera wyjsciowego
	InFormTransporterBeforeScrewerErrorCode 						AT %I*:UINT;			(*po kom*)

	(*****************TRANSPORTER ZA ZAKRECARKAMI*******************)
	fbFormTransporterAfterScrewer									: FB_MitsubishiInverter;
	eFormTransporterAfterScrewerState								: E_Station;			
	eFormTransporterAfterScrewerRunningState						: E_ConveyorState;	
	fbFormTransporterAfterScrewerState								: FB_State;		
	QnFormTransporterAfterScrewerVelocitySV 						AT %Q*: UDINT; 			(*po kom*)	// Nastawa prędkości transportera
	InFormTransporterAfterScrewerVelocityCV 						AT %I*: UDINT;			(*po kom*)
	InFormTransporterAfterScrewerSTW 								AT %I*: UINT; 			(*po kom*)	// Statusword transportera wyjściowego
	QnFormTransporterAfterScrewerCTW 								AT %Q*: UINT;  			(*po kom*)	// Controlword transportera wyjsciowego
	InFormTransporterAfterScrewerErrorCode 							AT %I*:UINT;			(*po kom*)

	(*Smieci*)
	bConveyorTest1											: BOOL;
	bConveyorTest2											: BOOL;
	bConveyorTest3											: BOOL;
	
	(*inne*)
	
	bConveyorTest4: BOOL;
		bConveyorTest5: BOOL;
END_VAR

aFormTransporterConveyor();
(*
eFormTransporterDispencerRunningState						:=eFormTransporterDispencerState;
eFormTransporterScrewerRunningState							:=eFormTransporterScrewerState;
eFormTransporterSlowerRunningState							:=eFormTransporterSlowerState;
*)

(********* GENEROWANIE STANU STACJI DO WIZKI**********)
fbFormTransporterDispencerState(
	eState													:= eFormTransporterDispencerState , 
	bRun													:= bFormTransportersDispencerCmdStart OR VIS.bFormTransporterDispencerManualCmdStart,	
	eConveyorRunningState									:= eFormTransporterDispencerRunningState , 
	sStateDesc												=> VIS.sFormTransporterDispencerState,
	iState													=>VIS.iFormTransporterDispencerState	);
	
fbFormTransporterScrewerState(
	eState													:= eFormTransporterScrewerState , 
	bRun													:= bFormTransportersScrewerCmdStart OR VIS.bFormTransporterScrewerManualCmdStart,	
	eConveyorRunningState									:= eFormTransporterScrewerRunningState	 , 
	sStateDesc												=> VIS.sFormTransporterScrewerState,
	iState													=> VIS.iFormTransporterScrewerState	);	
	
fbFormTransporterBeforeScrewerState(
	eState													:= eFormTransporterBeforeScrewerState , 
	bRun													:= bFormTransportersBeforeScrewerCmdStart OR VIS.bFormTransporterBeforeScrewerManualCmdStart,	
	eConveyorRunningState									:= eFormTransporterBeforeScrewerRunningState , 
	sStateDesc												=> VIS.sFormTransporterBeforeScrewerState,
	iState													=> VIS.iFormTransporterBeforeScrewerState	);	
	
	
(***** KONIEC GENEROWANIE STANU STACJI DO WIZKI*******)


VIS.nFormTransporterDispencerVelocityCV		:=	UDINT_TO_INT(InFormTransporterDispencerVelocityCV);
VIS.nFormTransporterScrewerVelocityCV 		:=	UDINT_TO_INT(InFormTransporterScrewerVelocityCV);
VIS.nFormTransporterBeforeScrewerVelocityCV	:=	UDINT_TO_INT(InFormTransporterBeforeScrewerVelocityCV);

ACTION aFormTransporterConveyor:
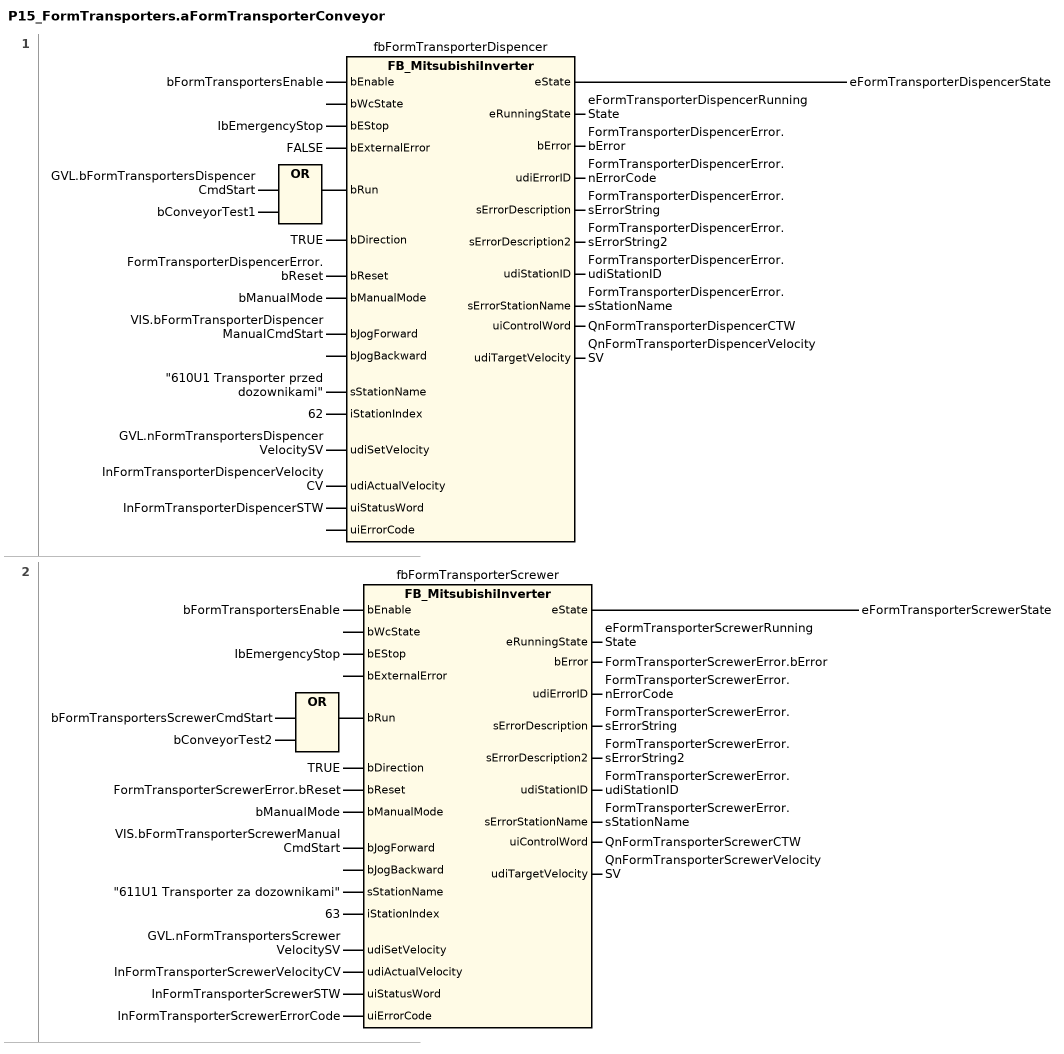
// NETWORK 1
fbFormTransporterDispencer(
    bEnable := bFormTransportersEnable,
    bEStop := IbEmergencyStop,
    bExternalError := FALSE,
    bRun := GVL.bFormTransportersDispencerCmdStart OR bConveyorTest1,
    bDirection := TRUE,
    bReset := FormTransporterDispencerError.bReset,
    bManualMode := bManualMode,
    bJogForward := VIS.bFormTransporterDispencerManualCmdStart,
    sStationName := "610U1 Transporter przed dozownikami",
    iStationIndex := 62,
    udiSetVelocity := GVL.nFormTransportersDispencerVelocitySV,
    udiActualVelocity := InFormTransporterDispencerVelocityCV,
    uiStatusWord := InFormTransporterDispencerSTW,
    eRunningState => eFormTransporterDispencerRunningState,
    bError => FormTransporterDispencerError.bError,
    udiErrorID => FormTransporterDispencerError.nErrorCode,
    sErrorDescription => FormTransporterDispencerError.sErrorString,
    sErrorDescription2 => FormTransporterDispencerError.sErrorString2,
    udiStationID => FormTransporterDispencerError.udiStationID,
    sErrorStationName => FormTransporterDispencerError.sStationName,
    uiControlWord => QnFormTransporterDispencerCTW,
    udiTargetVelocity => QnFormTransporterDispencerVelocitySV); // FB_MitsubishiInverter
eFormTransporterDispencerState := fbFormTransporterDispencer.eState;

// NETWORK 2
fbFormTransporterScrewer(
    bEnable := bFormTransportersEnable,
    bEStop := IbEmergencyStop,
    bRun := bFormTransportersScrewerCmdStart OR bConveyorTest2,
    bDirection := TRUE,
    bReset := FormTransporterScrewerError.bReset,
    bManualMode := bManualMode,
    bJogForward := VIS.bFormTransporterScrewerManualCmdStart,
    sStationName := "611U1 Transporter za dozownikami",
    iStationIndex := 63,
    udiSetVelocity := GVL.nFormTransportersScrewerVelocitySV,
    udiActualVelocity := InFormTransporterScrewerVelocityCV,
    uiStatusWord := InFormTransporterScrewerSTW,
    uiErrorCode := InFormTransporterScrewerErrorCode,
    eRunningState => eFormTransporterScrewerRunningState,
    bError => FormTransporterScrewerError.bError,
    udiErrorID => FormTransporterScrewerError.nErrorCode,
    sErrorDescription => FormTransporterScrewerError.sErrorString,
    sErrorDescription2 => FormTransporterScrewerError.sErrorString2,
    udiStationID => FormTransporterScrewerError.udiStationID,
    sErrorStationName => FormTransporterScrewerError.sStationName,
    uiControlWord => QnFormTransporterScrewerCTW,
    udiTargetVelocity => QnFormTransporterScrewerVelocitySV); // FB_MitsubishiInverter
eFormTransporterScrewerState := fbFormTransporterScrewer.eState;

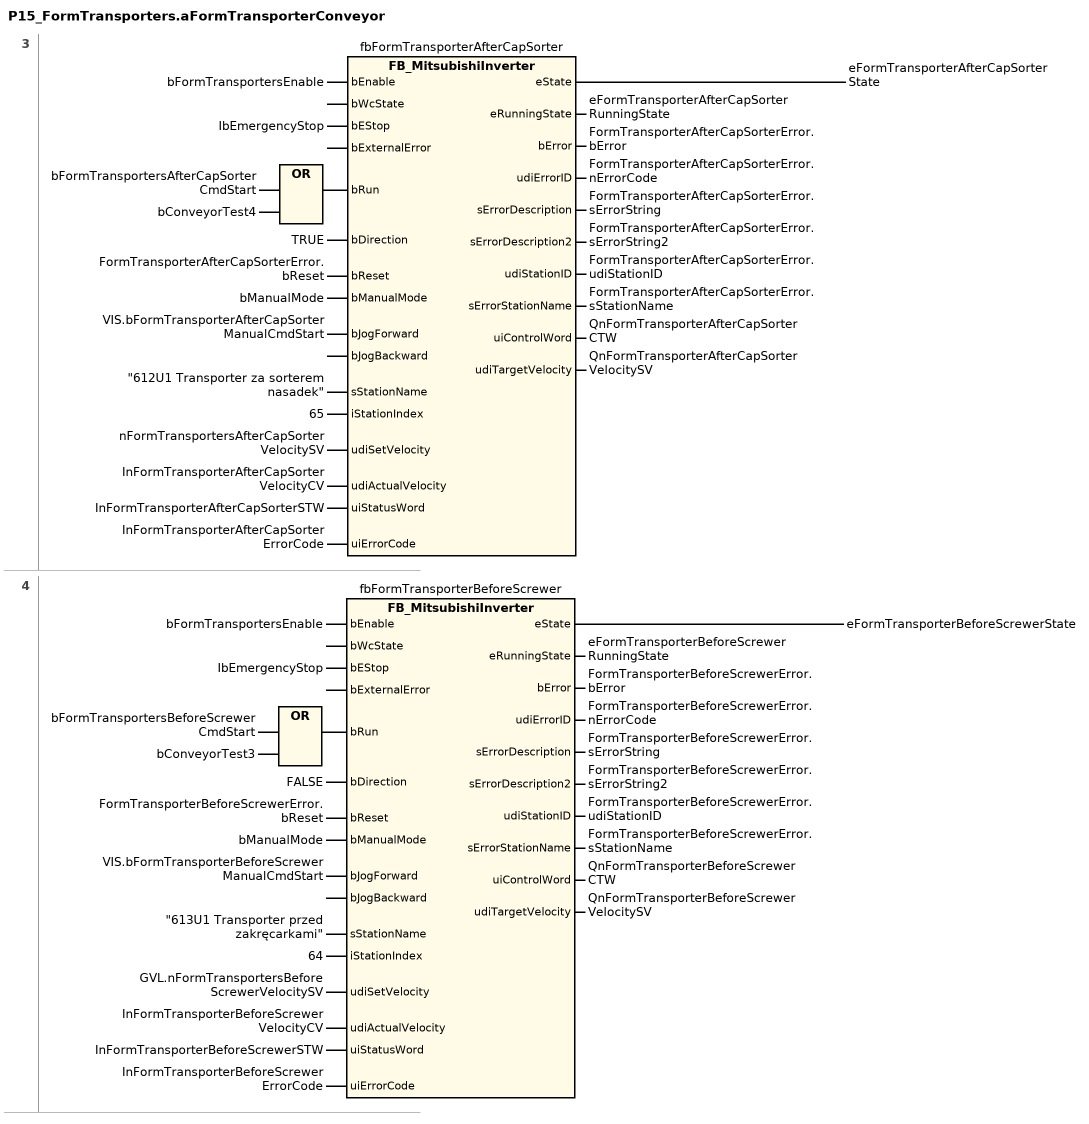
// NETWORK 3
fbFormTransporterAfterCapSorter(
    bEnable := bFormTransportersEnable,
    bEStop := IbEmergencyStop,
    bRun := bFormTransportersAfterCapSorterCmdStart OR bConveyorTest4,
    bDirection := TRUE,
    bReset := FormTransporterAfterCapSorterError.bReset,
    bManualMode := bManualMode,
    bJogForward := VIS.bFormTransporterAfterCapSorterManualCmdStart,
    sStationName := "612U1 Transporter za sorterem nasadek",
    iStationIndex := 65,
    udiSetVelocity := nFormTransportersAfterCapSorterVelocitySV,
    udiActualVelocity := InFormTransporterAfterCapSorterVelocityCV,
    uiStatusWord := InFormTransporterAfterCapSorterSTW,
    uiErrorCode := InFormTransporterAfterCapSorterErrorCode,
    eRunningState => eFormTransporterAfterCapSorterRunningState,
    bError => FormTransporterAfterCapSorterError.bError,
    udiErrorID => FormTransporterAfterCapSorterError.nErrorCode,
    sErrorDescription => FormTransporterAfterCapSorterError.sErrorString,
    sErrorDescription2 => FormTransporterAfterCapSorterError.sErrorString2,
    udiStationID => FormTransporterAfterCapSorterError.udiStationID,
    sErrorStationName => FormTransporterAfterCapSorterError.sStationName,
    uiControlWord => QnFormTransporterAfterCapSorterCTW,
    udiTargetVelocity => QnFormTransporterAfterCapSorterVelocitySV); // FB_MitsubishiInverter
eFormTransporterAfterCapSorterState := fbFormTransporterAfterCapSorter.eState;

// NETWORK 4
fbFormTransporterBeforeScrewer(
    bEnable := bFormTransportersEnable,
    bEStop := IbEmergencyStop,
    bRun := bFormTransportersBeforeScrewerCmdStart OR bConveyorTest3,
    bDirection := FALSE,
    bReset := FormTransporterBeforeScrewerError.bReset,
    bManualMode := bManualMode,
    bJogForward := VIS.bFormTransporterBeforeScrewerManualCmdStart,
    sStationName := "613U1 Transporter przed zakręcarkami",
    iStationIndex := 64,
    udiSetVelocity := GVL.nFormTransportersBeforeScrewerVelocitySV,
    udiActualVelocity := InFormTransporterBeforeScrewerVelocityCV,
    uiStatusWord := InFormTransporterBeforeScrewerSTW,
    uiErrorCode := InFormTransporterBeforeScrewerErrorCode,
    eRunningState => eFormTransporterBeforeScrewerRunningState,
    bError => FormTransporterBeforeScrewerError.bError,
    udiErrorID => FormTransporterBeforeScrewerError.nErrorCode,
    sErrorDescription => FormTransporterBeforeScrewerError.sErrorString,
    sErrorDescription2 => FormTransporterBeforeScrewerError.sErrorString2,
    udiStationID => FormTransporterBeforeScrewerError.udiStationID,
    sErrorStationName => FormTransporterBeforeScrewerError.sStationName,
    uiControlWord => QnFormTransporterBeforeScrewerCTW,
    udiTargetVelocity => QnFormTransporterBeforeScrewerVelocitySV); // FB_MitsubishiInverter
eFormTransporterBeforeScrewerState := fbFormTransporterBeforeScrewer.eState;

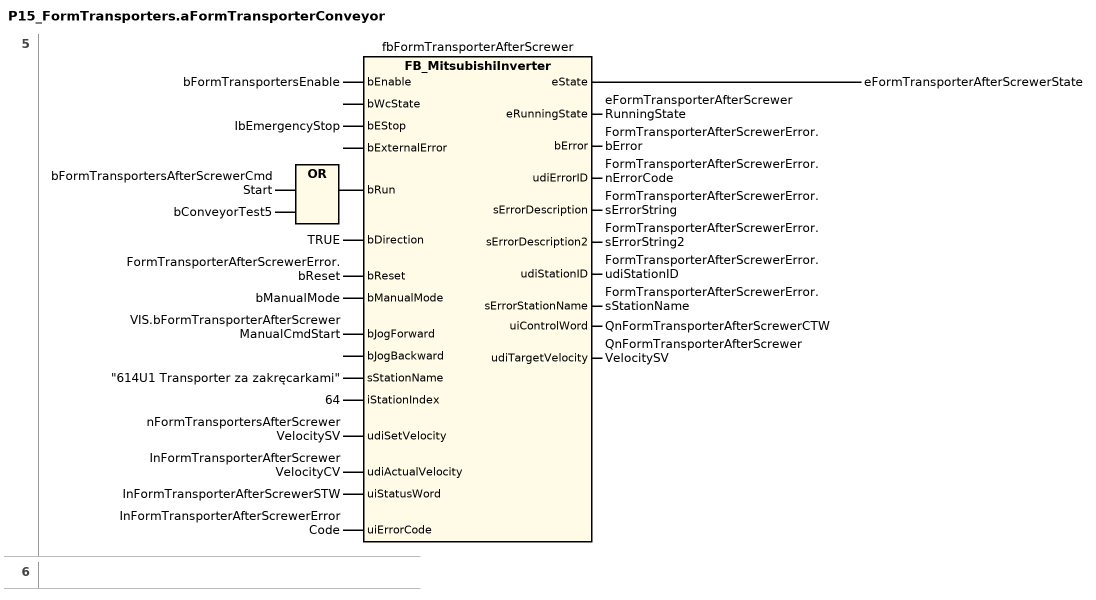
// NETWORK 5
fbFormTransporterAfterScrewer(
    bEnable := bFormTransportersEnable,
    bEStop := IbEmergencyStop,
    bRun := bFormTransportersAfterScrewerCmdStart OR bConveyorTest5,
    bDirection := TRUE,
    bReset := FormTransporterAfterScrewerError.bReset,
    bManualMode := bManualMode,
    bJogForward := VIS.bFormTransporterAfterScrewerManualCmdStart,
    sStationName := "614U1 Transporter za zakręcarkami",
    iStationIndex := 64,
    udiSetVelocity := nFormTransportersAfterScrewerVelocitySV,
    udiActualVelocity := InFormTransporterAfterScrewerVelocityCV,
    uiStatusWord := InFormTransporterAfterScrewerSTW,
    uiErrorCode := InFormTransporterAfterScrewerErrorCode,
    eRunningState => eFormTransporterAfterScrewerRunningState,
    bError => FormTransporterAfterScrewerError.bError,
    udiErrorID => FormTransporterAfterScrewerError.nErrorCode,
    sErrorDescription => FormTransporterAfterScrewerError.sErrorString,
    sErrorDescription2 => FormTransporterAfterScrewerError.sErrorString2,
    udiStationID => FormTransporterAfterScrewerError.udiStationID,
    sErrorStationName => FormTransporterAfterScrewerError.sStationName,
    uiControlWord => QnFormTransporterAfterScrewerCTW,
    udiTargetVelocity => QnFormTransporterAfterScrewerVelocitySV); // FB_MitsubishiInverter
eFormTransporterAfterScrewerState := fbFormTransporterAfterScrewer.eState;

// NETWORK 6
END_ACTION

END_PROGRAM

// ---- POUs/P00_Signalization.TcPOU
(*
Nazwa:			P00_Signalization
Opis:			Sygnalizacja na lini
Wersja:			v0.1
Data:			2018-10-10
Autor:			DP
Urzadzenia:		
Konfiguracja:	
Info:

*)
PROGRAM P00_Signalization
VAR

	QiLineRedSignalizationLamp 		AT %Q*:INT;				// Sygnalizacja czerwony kolor listwy LED
	QiLineGreenSignalizationLamp 	AT %Q*:INT;				// Sygnalizacja zielony kolor listwy LED	
	QiLineBlueSignalizationLamp 	AT %Q*:INT;				// Sygnalizacja niebieski kolor listwy LED		
	QiLineWhiteSignalizationLamp 	AT %Q*:INT;				// Sygnalizacja biały kolor listwy LED	
	                                            			
	QbStartLamp			 			AT %Q*:BOOL;				// Sygnalizacja startu cyklu poprzez lampkę na przyciskac
	QbResetLamp 					AT %Q*:BOOL; 				// Sygnalizacja Resetu bezpieczeństwa poprzez lampkę naprzycisku reset
	QbBuzzer						AT %Q*:BOOL;	

	QbTurnTableStartLamp			AT %Q*:BOOL;				// Sygnalizacja startu cyklu poprzez lampkę na przyciskac		
	QbTurnTableResetLamp			AT %Q*:BOOL; 				// Sygnalizacja Resetu bezpieczeństwa poprzez lampkę naprzycisku reset

	QbPucksInserterStartLamp		AT %Q*:BOOL;				// Sygnalizacja startu cyklu poprzez lampkę na przyciskac		
	QbPucksInserterResetLamp		AT %Q*:BOOL; 				// Sygnalizacja Resetu bezpieczeństwa poprzez lampkę naprzycisku reset

	
	(**BottleTransfer****)
//	QbBottleTransferRedSignalizationLamp AT %Q*:BOOL;		(*PLC.G1 robot*)		// Sygnalizacja czerwony kolor listwy LED
//	QbBottleTransferGreenSignalizationLamp AT %Q*:BOOL;		(*PLC.G1 robot*)		// Sygnalizacja zielony kolor listwy LED	
//	QbBottleTransferBlueSignalizationLamp AT %Q*:BOOL;		(*PLC.G1 robot*)		// Sygnalizacja niebieski kolor listwy LED		
//	QbBottleTransferWhiteSignalizationLamp AT %Q*:BOOL;		(*PLC.G1 robot*)		// Sygnalizacja biały kolor listwy LED	
		
	rtErrorOccure: R_TRIG;
	tofrtErrorOccure: TOF;
	TimerServiceMode: TON;
	
	
	fb1HzBlink : FB_Blink_S; // Blok wykorzystywany do wymigiwania lampki resetu
	fb5HzBlink : FB_Blink_S; // Blok wykorzystywany do wymigiwania lampki resetu
	
	
	//FB's taśma RGB
	fbRgbLedTape				: FB_RgbLedTape_EL2563;	//DMX Ul (górna taśma)
	
	//Kolor taśma LED RGB
	fbPackMlToRgb				: FB_PackMlToRgb_EL2564;//Conwersja PackML Ul w colory RGB i tryb pracy dla taśmy górnej w UL50
	
	eLastState					: E_PackMLState;
	eLastStateTemp				: E_PackMLState;
	AiProcessData				: ARRAY [1..5] OF INT;
	
	 iStep : INT := 0; // Aktualny krok efektu
    iTimer : TON; // Timer dla opóźnienia między efektami
    bTimerElapsed : BOOL := FALSE; // Flaga wskazująca, że czas minął
    iBrightness : INT := 0; // Jasność (dla efektu pulsowania)
    bIncreasing : BOOL := TRUE; // Flaga wskazująca kierunek zmiany jasności
	bTestLed: BOOL;
 	iNoteIndex : INT := 0; 
    iTimer2 : TON; 
    bTimerElapsed2 : BOOL := FALSE; 
    iDuration : TIME := T#0MS; 
    iFrequency : INT := 0; 
	
    arrM : ARRAY[1..19] OF INT := [440, 440, 440, 349, 440, 349, 440, 0, 440, 440, 440, 349, 440, 349, 440, 0, 440, 440, 440];
    arrDuration : ARRAY[1..19] OF TIME := [T#500MS, T#500MS, T#500MS, T#350MS, T#500MS, T#350MS, T#1000MS, 
                                           T#500MS, T#500MS, T#500MS, T#500MS, T#350MS, T#500MS, T#350MS, T#1000MS, 
                                           T#500MS, T#500MS, T#500MS, T#500MS];
    iMLength : INT := 19; 
	
END_VAR

(*sygnalizacja główna*)
aLamps();

ACTION aLamps:
fb1HzBlink(Tv:=T#1S);
fb5HzBlink(Tv:=T#200MS);


(*****Listwy LED*****)
(*QiLineRedSignalizationLamp:=VIS.bErrorOccure OR P00_PackML.fbPMLAuto.ePMLState = E_PMLState.ePMLState_ABORTED OR VIS.bRecipeWizardOn;
QiLineGreenSignalizationLamp:=(b2Hz AND P00_PackML.fbPMLAuto.ePMLState = E_PMLState.ePMLState_STARTING ) OR (VIS.bRecipeWizardOn AND NOT (VIS.bErrorOccure)) OR P00_PackML.fbPMLAuto.ePMLState = E_PMLState.ePMLState_STARTING OR P00_PackML.fbPMLAuto.ePMLState = E_PMLState.ePMLState_EXECUTE;
//Sterowanie Niebieskim światłem listwy led
TimerServiceMode(IN:=P00_PackML.fbPMLAuto.ePMLState = E_PMLState.ePMLState_IDLE AND P00_PackML.fbServiceMode.bOut,PT:=T#5S);
QiLineBlueSignalizationLamp:= P00_PackML.fbPMLAuto.ePMLState = E_PMLState.ePMLState_IDLE AND NOT VIS.bRecipeWizardOn AND P00_PackML.fbServiceMode.bOut;
QiLineWhiteSignalizationLamp:= (NOT QiLineRedSignalizationLamp) AND (NOT QiLineBlueSignalizationLamp) AND (NOT QiLineGreenSignalizationLamp) AND NOT VIS.bRecipeWizardOn AND NOT (P00_PackML.fbPMLAuto.ePMLState = E_PMLState.ePMLState_EXECUTE); 
*)
//Vasyl 03.10 Reset nie mruga póki nie skończy się timer tonbFirstCycle.Q w ACT_SafetyFirstResetDelay
(*****Przyciski*****)
QbStartLamp := (((	P00_PackML.fbPMLAuto.ePMLState = Tc3_PackML.E_PMLState.ePMLState_IDLE  OR P00_PackML.fbPMLAuto.ePMLState = Tc3_PackML.E_PMLState.ePMLState_SUSPENDED) AND 
               		P00_PackML.fbPMLModeManager.eModeStatus = Tc3_PackML.E_PMLUnitMode.ePMLUnitMode_AUTOMATIC AND (P00_PackML.bStationsAreReady AND NOT P00_PackML.bAtLeastOneOfTheStationsNeedHoming)) AND fb1HzBlink.Q);
			   
QbResetLamp:=NOT IbEmergencyStop AND b1Hz AND P00_PackML.tonbFirstCycle.Q;

QbTurnTableStartLamp	:=	QbStartLamp;
QbTurnTableResetLamp	:=	QbResetLamp;

QbPucksInserterStartLamp:=	QbStartLamp;
QbPucksInserterResetLamp:=	QbResetLamp;

(*****Buzzer********)
rtErrorOccure 			(CLK :=VIS.bErrorOccure, Q=>);
tofrtErrorOccure 		(IN := rtErrorOccure.Q , PT := T#5S);
IF NOT bTestLed THEN
QbBuzzer 			:=	(P00_PackML.fbPMLAuto.ePMLState = Tc3_PackML.E_PMLState.ePMLState_STARTING AND b1Hz AND NOT P00_PackML.tonStarting.Q) OR bSoftAlarm OR (tofrtErrorOccure.Q AND b1Hz);
END_IF

(*Warningi*)
IF (P08_CapFeeder.fbCapFeeder.bWarning1 OR P01_BottleFeeder.fbBottleFeeder.bWarning1) AND P00_PackML.fbPMLAuto.ePMLState = Tc3_PackML.E_PMLState.ePMLState_EXECUTE THEN
	(*QiLineRedSignalizationLamp			:= TRUE;
	QiLineGreenSignalizationLamp			:= FALSE;
	QiLineBlueSignalizationLamp				:= TRUE;
	QiLineWhiteSignalizationLamp			:= FALSE;*)
END_IF


IF VIS.bWeighingForm AND b1Hz AND P00_PackML.fbPMLAuto.ePMLState = Tc3_PackML.E_PMLState.ePMLState_EXECUTE THEN
	(*QiLineRedSignalizationLamp				:= FALSE; 
	QiLineGreenSignalizationLamp			:= TRUE;
	QiLineBlueSignalizationLamp				:= TRUE;
	QiLineWhiteSignalizationLamp			:= FALSE;*)
END_IF


fbPackMlToRgb(
					ePackMLState		:= P00_PackML.fbPMLAuto.ePMLState,
					ePackMLMode			:= P00_PackML.fbPMLModeManager.eModeStatus, 
					eLastState			:= eLastState, 
					nDelayButtonBlinkIn	:= , 
					bStopViaOut			:= , 
					bWarning			:= VIS.uliWarningOccure>0, 
					bHoming				:= Gvl.bHoming, 
					bWeighingForm		:= VIS.bWeighingForm,
					bLowMaterialInExecute:=	P00_Visualization.tonNoFormsBeforeDispencers.Q OR 
											P00_PackML.tonCycleBadBottleConveyorFullSensor.Q OR P16_LabelMachine.tonLabelMachineFullSensorInfo.Q OR
											P06_LidFeeder.bLidFeederWarning1 OR P06_LidFeeder.bLidFeederWarning2 OR
											P06_WickFeeder.fbWickFeederSt.bWarning,
					nCh1Red				=> ,
					nCh2Green			=> ,
					nCh3Blue			=> , 
					nCh4White			=> , 
					nCh5Reserve=> , 
					bBlink=> , 
					bBlink2Colors=> , 					
					bHorn=> , 
					bStartButtonLampOut=> );

fbRgbLedTape(	 
				   	bEnable				:= TRUE,
					nCh1Red				:= fbPackMlToRgb.nCh1Red,
					nCh2Green			:= fbPackMlToRgb.nCh2Green,
					nCh3Blue			:= fbPackMlToRgb.nCh3Blue,
					nCh4White			:= fbPackMlToRgb.nCh4White,
					nCh5Reserve			:= fbPackMlToRgb.nCh5Reserve,
					bBlink				:= fbPackMlToRgb.bBlink,
					bBlink2Colors		:= fbPackMlToRgb.bBlink2Colors,					
					nDelayBlink 		:= 1,
					nMaxBlinkValue		:= 32766,
					AiProcessData		:= AiProcessData);
IF NOT bTestLed THEN		
	QiLineRedSignalizationLamp 				:= AiProcessData[1];  
	QiLineGreenSignalizationLamp 			:= AiProcessData[2];
	QiLineBlueSignalizationLamp 			:= AiProcessData[3];
	QiLineWhiteSignalizationLamp 			:= AiProcessData[4];
ELSE
		// Logika sterowania
	iTimer(IN := TRUE, PT := T#500MS); // Timer ustawiony na 500 ms
	bTimerElapsed := iTimer.Q;
	
	IF bTimerElapsed THEN
		iTimer(IN := FALSE); // Resetowanie timera
		iTimer(IN := TRUE);  // Restart timera
		
		CASE iStep OF
			0: // Czerwony
				QiLineRedSignalizationLamp := 10000; // Maksymalna jasność
				QiLineGreenSignalizationLamp := 0;
				QiLineBlueSignalizationLamp := 0;
				QiLineWhiteSignalizationLamp := 0;
			1: // Zielony
				QiLineRedSignalizationLamp := 0;
				QiLineGreenSignalizationLamp := 10000; // Maksymalna jasność
				QiLineBlueSignalizationLamp := 0;
				QiLineWhiteSignalizationLamp := 0;
			2: // Niebieski
				QiLineRedSignalizationLamp := 0;
				QiLineGreenSignalizationLamp := 0;
				QiLineBlueSignalizationLamp := 10000; // Maksymalna jasność
				QiLineWhiteSignalizationLamp := 0;
			3: // Biały
				QiLineRedSignalizationLamp := 0;
				QiLineGreenSignalizationLamp := 0;
				QiLineBlueSignalizationLamp := 0;
				QiLineWhiteSignalizationLamp := 10000; // Maksymalna jasność
			4: // Pulsowanie jasności
				IF bIncreasing THEN
					iBrightness := iBrightness + 1000;
					IF iBrightness >= 10000 THEN
						bIncreasing := FALSE;
					END_IF
				ELSE
					iBrightness := iBrightness - 1000;
					IF iBrightness <= 0 THEN
						bIncreasing := TRUE;
					END_IF
				END_IF
				QiLineRedSignalizationLamp := iBrightness;
				QiLineGreenSignalizationLamp := iBrightness;
				QiLineBlueSignalizationLamp := iBrightness;
				QiLineWhiteSignalizationLamp := iBrightness;
		END_CASE;
		
		iStep := iStep + 1;
		IF iStep > 4 THEN
			iStep := 0; // Powrót do pierwszego kroku
		END_IF;
	END_IF;
	
    // Timer nuty
    iTimer2(IN := TRUE, PT := iDuration); 
    bTimerElapsed2 := iTimer2.Q;

    IF bTimerElapsed2 THEN

        iTimer2(IN := FALSE); // Reset timera
        iTimer2(IN := TRUE);  // Restart timera
        iNoteIndex := iNoteIndex + 1;
       
        IF iNoteIndex > iMLength THEN
            iNoteIndex := 1;
        END_IF;

        // Ustawienie częstotliwości i czasu trwania 
        iFrequency := arrM[iNoteIndex];
        iDuration := arrDuration[iNoteIndex];

        // Generowanie dźwięku na buzzerze
        IF iFrequency > 0 THEN
            QbBuzzer := TRUE; // Aktywacja buzzera
        ELSE
            QbBuzzer := FALSE; // Pauza
        END_IF;
    END_IF;	
		
END_IF

(*
fbRgbLedTape(	 
				   	bEnable				:= TRUE,
					nCh1Red				:= 0,
					nCh2Green			:= 32000,
					nCh3Blue			:= 10000,
					nCh4White			:= 0,
					nCh5Reserve			:= 0,
					bBlink				:= FALSE,
					bBlink2Colors		:= TRUE,					
					nDelayBlink 		:= 1,
					nMaxBlinkValue		:= 32766,
					AiProcessData		:= AiProcessData);
			
QiLineRedSignalizationLamp 				:= 	AiProcessData[1];
QiLineGreenSignalizationLamp 			:= 	AiProcessData[2];
QiLineBlueSignalizationLamp 			:= 	AiProcessData[3];
QiLineWhiteSignalizationLamp 			:= 	AiProcessData[4];
*)
END_ACTION

END_PROGRAM

// ---- POUs/FB/Blinkers/FB_Blink_S.TcPOU
(********************************************************************************************)
(*							Beckhoff Automation Poland										*)
(*								FB_Blink_S	 v1.1											*)
(*									9.11.2007												*)
(*						Blok funkcyjny zegara synchronicznego								*)
(*__________________________________________________________________________________________*)

FUNCTION_BLOCK FB_Blink_S
VAR_INPUT
	Tv										:	TIME;				(*Czas trwania impulsu i przerwy*)
END_VAR
VAR_OUTPUT
	Q										:	BOOL;				(*Wyjscie*)
END_VAR
VAR
	ton1									:	TON;
	ton2									:	TON;
END_VAR

ton1(IN:= NOT ton2.Q, PT:=Tv);
Q:=ton1.Q;
ton2(IN:=ton1.Q , PT:=ton1.PT );

END_FUNCTION_BLOCK

// ---- POUs/FB/Led/FB_RgbLedTape_EL2563.TcPOU
(*
Nazwa:			FB_RgbLedTape
Opis:			Sterowanie taśmamy przez moduł sterownika EL6851
Wersja:			v0.2
Data:			2024-03-13
Autor:			AM,DP
Urzadzenia:		EL6851
Konfiguracja:	GVL_DMX z aProcessData
Info:
Zmiany:
- 20240318 [DP] Dodanie migajacych dwóch kolorów na przemian
*)
FUNCTION_BLOCK FB_RgbLedTape_EL2563

VAR_INPUT
	
	bEnable					:		BOOL;	
	nCh1Red					:		INT;
	nCh2Green				:		INT;
	nCh3Blue				:		INT;
	nCh4White				:		INT;
	nCh5Reserve				:		INT;
	
	bBlink					:		BOOL;
	bBlink2Colors			:		BOOL;	
	nDelayBlink				:		INT :=5;
	nMaxBlinkValue			:		INT:=16000;	

	nMinBlinkValue			:		INT:=2000;	
END_VAR

VAR_OUTPUT
END_VAR

VAR_IN_OUT
	AiProcessData			   : ARRAY [1..5] OF INT;
END_VAR

VAR
	nCycleBlink			:	INT;	//Liczylnik cyklów dla tryby Migamie 
	nBlinkValue			:	INT;	//Biegle znaczenie dla migania
	bBlinkDir			:	BOOL; 	//kierunek (zmieńszenie/zwiękzenie nBlinkValue)
	bChangeColor: BOOL;
	iBlink2ColorsCase: INT;
	toniBlink2ColorsCase: TON;
END_VAR

IF (bEnable) THEN
	IF (bBlink2Colors) THEN
		actBlink2Colors();
	ELSIF (bBlink) THEN
		actBlink();
	ELSE
		actNoBlink();
	END_IF
	
	
END_IF

ACTION actBlink:
IF (nCh1Red>0) THEN
	AiProcessData[1] := nBlinkValue;
ELSE
	AiProcessData[1] := 0;
END_IF

IF (nCh2Green>0) THEN
	AiProcessData[2] := nBlinkValue;
ELSE
	AiProcessData[2] := 0;
END_IF
	
IF (nCh3Blue>0) THEN
	AiProcessData[3] := nBlinkValue;
ELSE
	AiProcessData[3] := 0;
END_IF

IF (nCh4White>0) THEN
	AiProcessData[4] := nBlinkValue;
ELSE
	AiProcessData[4] := 0;
END_IF

IF (nCh5Reserve>0) THEN
	AiProcessData[5] := nBlinkValue;
ELSE
	AiProcessData[5] := 0;
END_IF

//Inc/dec dla nBlinkValue
nCycleBlink := nCycleBlink + 1;
IF (nCycleBlink > nDelayBlink) THEN
	
	//dodac
	IF (nBlinkValue < nMaxBlinkValue AND NOT bBlinkDir) THEN
		nBlinkValue :=nBlinkValue + 50;
		IF nBlinkValue < 0 THEN
		nBlinkValue := nMaxBlinkValue;
		bBlinkDir := TRUE;
		END_IF
	ELSE
		bBlinkDir := TRUE;
	END_IF
	
	//zwiększyć
	IF (nBlinkValue > nMinBlinkValue AND bBlinkDir) THEN
		nBlinkValue :=nBlinkValue - 100;
		IF nBlinkValue < 0 THEN
		nBlinkValue := nMinBlinkValue;
		bBlinkDir := FALSE;
		END_IF
	ELSE
		bBlinkDir := FALSE;
	END_IF
	
	nCycleBlink :=0;
END_IF
END_ACTION

ACTION actBlink2Colors:
bChangeColor;
toniBlink2ColorsCase(IN:=iBlink2ColorsCase=50,PT:=T#100MS);
CASE iBlink2ColorsCase OF
	0:
		AiProcessData[1] 	:= 0;
		AiProcessData[2] 	:= nCh2Green;
		AiProcessData[3] 	:= 0;
		AiProcessData[4] 	:= 0;
		
		iBlink2ColorsCase	:=	iBlink2ColorsCase	+	10;
		
	10:
		AiProcessData[2] := 	AiProcessData[2] - 50;
		IF 	AiProcessData[2] < 100 THEN
			iBlink2ColorsCase	:=	iBlink2ColorsCase	+	10;
		END_IF
		
	20:
		AiProcessData[3] 	:= 	AiProcessData[3] + 100;
		IF 	AiProcessData[3] > 32000 THEN
			iBlink2ColorsCase	:=	iBlink2ColorsCase	+	10;
		END_IF	

	30:
		AiProcessData[3] 	:= 	AiProcessData[3] - 100;
		IF 	AiProcessData[3] < 200 THEN
			iBlink2ColorsCase	:=	iBlink2ColorsCase	+	10;
		END_IF	
	
	40:
		AiProcessData[2] := 	AiProcessData[2] + 50;
		IF 	AiProcessData[2] > nCh2Green THEN
			iBlink2ColorsCase	:=	iBlink2ColorsCase	+	10;
		END_IF		
		
	50:
		IF toniBlink2ColorsCase.Q THEN
			iBlink2ColorsCase	:=	0;
		END_IF
END_CASE
END_ACTION

ACTION actNoBlink:
AiProcessData[1] :=nCh1Red;
AiProcessData[2] :=nCh2Green;
AiProcessData[3] :=nCh3Blue;
AiProcessData[4] :=nCh4White;
AiProcessData[5] :=nCh5Reserve;
END_ACTION

END_FUNCTION_BLOCK

// ---- POUs/FB/Led/FB_PackMlToRgb_EL2564.TcPOU
(*
Nazwa:			FB_PackMlToRgb
Opis:			Konwersja PackML statr w colory RGB i tryb pracy taśmy (dla standartowych taśm)
Wersja:			v0.2
Data:			2024-03-13
Autor:			AM,DP
Urzadzenia:		
Konfiguracja:	
Info:
Zmiany:
- 20240312 [DP] Przewazanie
*)
FUNCTION_BLOCK FB_PackMlToRgb_EL2564
VAR_INPUT
	ePackMLState					: E_PackMLState;
	ePackMLMode						: E_PackMLMode;
	eLastState						: E_PackMLState;
	
	nDelayButtonBlinkIn				: INT :=5;
	bStopViaOut						: BOOL;
	bWarning						: BOOL;
	bHoming							: BOOL;
	bWeighingForm					: BOOL;
	bLowMaterialInExecute			: BOOL;
END_VAR
VAR_OUTPUT
	nCh1Red							: INT;
	nCh2Green						: INT;
	nCh3Blue						: INT;
	nCh4White						: INT;
	nCh5Reserve						: INT;
	bBlink							: BOOL;	
	bBlink2Colors					: BOOL;		
	bHorn							: BOOL;
	bStartButtonLampOut				: BOOL;
END_VAR
VAR
	nCycleBlink						: INT;	//Liczylnik cyklów dla tryby Migamie 
	bStartButtonLamp				: BOOL;

END_VAR

actMain();

ACTION actButtonLamp:
IF (bStartButtonLamp) THEN
	nCycleBlink := nCycleBlink + 1;
	IF (nCycleBlink > nDelayButtonBlinkIn) THEN
		nCycleBlink :=0;
		bStartButtonLampOut := NOT bStartButtonLampOut;
	END_IF

ELSE
	bStartButtonLampOut	:=FALSE;
	nCycleBlink :=0;
END_IF
END_ACTION

ACTION actMain:
CASE ePackMLState OF
	
	E_PackMLState.eAborting:
		nCh1Red				:=32000;
		nCh2Green			:=0;
		nCh3Blue			:=0;
		nCh4White			:=0;
		nCh5Reserve			:=0;
		bBlink				:=TRUE;
		bBlink2Colors		:=FALSE;
		bStartButtonLamp	:=FALSE;
		bHorn				:=FALSE;
		
	E_PackMLState.eClearing:
		nCh1Red				:=32000;
		nCh2Green			:=0;
		nCh3Blue			:=0;
		nCh4White			:=0;
		nCh5Reserve			:=0;
		bBlink				:=FALSE;
		bBlink2Colors		:=FALSE;
		bStartButtonLamp	:=FALSE;
		bHorn				:=FALSE;
	
	E_PackMLState.eAborted:
		nCh1Red				:=32000;
		nCh2Green			:=0;
		nCh3Blue			:=0;
		nCh4White			:=0;
		nCh5Reserve			:=0;
		bBlink				:=TRUE;
		bBlink2Colors		:=FALSE;
		bStartButtonLamp	:=FALSE;
		bHorn				:=FALSE;


	E_PackMLState.eComplete:
		nCh1Red				:=0;
		nCh2Green			:=0;
		nCh3Blue			:=0;
		nCh4White			:=32000;
		nCh5Reserve			:=0;
		bBlink				:=FALSE;
		bBlink2Colors		:=FALSE;
		bStartButtonLamp	:=FALSE;
		bHorn				:=FALSE;

	E_PackMLState.eStopped:
		nCh1Red				:=32000;
		nCh2Green			:=0;
		nCh3Blue			:=0;
		nCh4White			:=0;
		nCh5Reserve			:=0;
		bBlink				:=FALSE;
			bBlink2Colors		:=FALSE;
		bStartButtonLamp	:=FALSE;
		bHorn				:=FALSE;
		
	E_PackMLState.eStopping:
	
		IF eLastState = E_PackMLState.eAborted OR eLastState = E_PackMLState.eClearing THEN
			nCh1Red				:=32000;
			nCh2Green			:=0;
			nCh3Blue			:=0;
			nCh4White			:=0;
			nCh5Reserve			:=0;
			bBlink				:=TRUE;
			bBlink2Colors		:=FALSE;
			bStartButtonLamp	:=FALSE;
			bHorn				:=FALSE;
		ELSE
			nCh1Red				:=0;
			nCh2Green			:=32000;
			nCh3Blue			:=0;
			nCh4White			:=0;
			nCh5Reserve			:=0;
			bBlink				:=TRUE;
			bBlink2Colors		:=FALSE;
			bStartButtonLamp	:=FALSE;
			bHorn				:=FALSE;
		END_IF
		
		
	E_PackMLState.eResetting:
		IF (NOT bHoming) THEN
			nCh1Red				:=32000;
			nCh2Green			:=0;
			nCh3Blue			:=0;
			nCh4White			:=0;
			nCh5Reserve			:=0;
			bBlink				:=TRUE;
			bBlink2Colors		:=FALSE;
			bStartButtonLamp	:=FALSE;
			bHorn				:=FALSE;
		ELSE				//Blekitny
			nCh1Red				:=0;
			nCh2Green			:=25000;
			nCh3Blue			:=32000;
			nCh4White			:=0;
			nCh5Reserve			:=0;
			bBlink				:=FALSE;
			bBlink2Colors		:=FALSE;
			bStartButtonLamp	:=FALSE;
			bHorn				:=FALSE;	
		END_IF

	E_PackMLState.eIdle:
		IF (NOT bHoming) THEN
		CASE ePackMLMode OF
			E_PackMLMode.eAutomatic:
				nCh1Red				:=0;
				nCh2Green			:=0;
				nCh3Blue			:=0;
				nCh4White			:=32000;
				nCh5Reserve			:=0;
				bBlink				:=FALSE;
				bBlink2Colors		:=FALSE;
				bStartButtonLamp	:=TRUE;
				bHorn				:=FALSE;
			E_PackMLMode.eManual:
				nCh1Red				:=0;
				nCh2Green			:=0;
				nCh3Blue			:=32000;
				nCh4White			:=0;
				nCh5Reserve			:=0;
				bBlink				:=FALSE;
				bBlink2Colors		:=FALSE;
				bStartButtonLamp	:=TRUE;
				bHorn				:=FALSE;
			E_PackMLMode.eMaintenance:
				nCh1Red				:=20000;
				nCh2Green			:=1000;
				nCh3Blue			:=32000;
				nCh4White			:=0;
				nCh5Reserve			:=0;
				bBlink				:=FALSE;
				bBlink2Colors		:=FALSE;
				bStartButtonLamp	:=TRUE;
				bHorn				:=FALSE;
			E_PackMLMode.eUndefined:
				nCh1Red				:=20000;
				nCh2Green			:=1000;
				nCh3Blue			:=32000;
				nCh4White			:=0;
				nCh5Reserve			:=0;
				bBlink				:=FALSE;
				bBlink2Colors		:=FALSE;
				bStartButtonLamp	:=TRUE;
				bHorn				:=FALSE;
		END_CASE
		ELSE
				nCh1Red				:=0;
				nCh2Green			:=32000;
				nCh3Blue			:=32000;
				nCh4White			:=0;
				nCh5Reserve			:=0;
				bBlink				:=FALSE;
				bBlink2Colors		:=FALSE;
				bStartButtonLamp	:=TRUE;
				bHorn				:=FALSE;	
		END_IF

	E_PackMLState.eStarting:
		nCh1Red				:=0;
		nCh2Green			:=32000;
		nCh3Blue			:=0;
		nCh4White			:=0;
		nCh5Reserve			:=0;
		bBlink				:=TRUE;
		bBlink2Colors		:=FALSE;
		bStartButtonLamp	:=FALSE;
		bHorn				:=TRUE;

	E_PackMLState.eExecute:
		IF bLowMaterialInExecute THEN
			nCh1Red				:=0;
			nCh2Green			:=32000;
			nCh3Blue			:=10000;
			nCh4White			:=0;
			nCh5Reserve			:=0;
			bBlink				:=FALSE;
			bBlink2Colors		:=TRUE;			
			bStartButtonLamp	:=FALSE;
			bHorn				:=FALSE;	
		ELSIF bWeighingForm THEN
			nCh1Red				:=0;
			nCh2Green			:=32000;
			nCh3Blue			:=32000;
			nCh4White			:=0;
			nCh5Reserve			:=0;
			bBlink				:=TRUE;
			bBlink2Colors		:=FALSE;
			bStartButtonLamp	:=FALSE;
			bHorn				:=FALSE;	
		ELSIF 	(bStopViaOut) THEN		//Różowy
			nCh1Red				:=32000;
			nCh2Green			:=0;
			nCh3Blue			:=16000;
			nCh4White			:=0;
			nCh5Reserve			:=0;
			bBlink				:=TRUE;
			bBlink2Colors		:=FALSE;
			bStartButtonLamp	:=FALSE;
			bHorn				:=FALSE;	
		ELSIF (NOT bWarning) THEN	//Zielony
			nCh1Red				:=0;
			nCh2Green			:=32000;
			nCh3Blue			:=0;
			nCh4White			:=0;
			nCh5Reserve			:=0;
			bBlink				:=FALSE;
			bBlink2Colors		:=FALSE;
			bStartButtonLamp	:=FALSE;
			bHorn				:=FALSE;
		ELSE						//Fioletowy
			nCh1Red				:=20000;
			nCh2Green			:=1000;
			nCh3Blue			:=32000;
			nCh4White			:=0;
			nCh5Reserve			:=0;
			bBlink				:=FALSE;
			bBlink2Colors		:=FALSE;
			bStartButtonLamp	:=FALSE;
			bHorn				:=FALSE;	
		END_IF
		
	E_PackMLState.eCompleting:
		nCh1Red				:=0;
		nCh2Green			:=32000;
		nCh3Blue			:=0;
		nCh4White			:=0;
		nCh5Reserve			:=0;
		bBlink				:=TRUE;
		bBlink2Colors		:=FALSE;
		bStartButtonLamp	:=FALSE;
		bHorn				:=FALSE;	
	
	E_PackMLState.eUnholding:
		nCh1Red				:=0;
		nCh2Green			:=32000;
		nCh3Blue			:=0;
		nCh4White			:=0;
		nCh5Reserve			:=0;
		bBlink				:=TRUE;
		bBlink2Colors		:=FALSE;
		bStartButtonLamp	:=FALSE;
		bHorn				:=TRUE;	

		
	E_PackMLState.eUnsuspending:
		nCh1Red				:=0;
		nCh2Green			:=32000;
		nCh3Blue			:=0;
		nCh4White			:=0;
		nCh5Reserve			:=0;
		bBlink				:=TRUE;
		bBlink2Colors		:=FALSE;
		bStartButtonLamp	:=FALSE;
		bHorn				:=TRUE;	

	E_PackMLState.eHolding:
		nCh1Red				:=0;
		nCh2Green			:=0;
		nCh3Blue			:=0;
		nCh4White			:=32000;
		nCh5Reserve			:=0;
		bBlink				:=TRUE;
		bBlink2Colors		:=FALSE;
		bStartButtonLamp	:=FALSE;
		bHorn				:=FALSE;
		
	E_PackMLState.eHeld:
		nCh1Red				:=0;
		nCh2Green			:=0;
		nCh3Blue			:=0;
		{warning ""}
		nCh4White			:=8000;
		nCh5Reserve			:=0;
		bBlink				:=FALSE;
		bBlink2Colors		:=FALSE;
		bStartButtonLamp	:=FALSE;
		bHorn				:=FALSE;
		
	E_PackMLState.eSuspending:
		nCh1Red				:=0;
		nCh2Green			:=0;
		nCh3Blue			:=0;
		nCh4White			:=32000;
		nCh5Reserve			:=0;
		bBlink				:=TRUE;
		bBlink2Colors		:=FALSE;
		bStartButtonLamp	:=FALSE;
		bHorn				:=FALSE;

	E_PackMLState.eSuspended:
		nCh1Red				:=0;
		nCh2Green			:=0;
		nCh3Blue			:=0;
		nCh4White			:=32000;
		nCh5Reserve			:=0;
		bBlink				:=FALSE;
		bBlink2Colors		:=FALSE;
		bStartButtonLamp	:=FALSE;
		bHorn				:=FALSE;
	
		
	E_PackMLState.eUndefined:
		nCh1Red				:=20000;
		nCh2Green			:=1000;
		nCh3Blue			:=32000;
		nCh4White			:=0;
		nCh5Reserve			:=0;
		bBlink				:=FALSE;
		bBlink2Colors		:=FALSE;
		bStartButtonLamp	:=FALSE;
		bHorn				:=FALSE;

		
	
		
	

		

		
	
	
		

		
	
		
	
		
	
		
	
		
	
		
	
END_CASE
END_ACTION

END_FUNCTION_BLOCK

// ---- POUs/P08_CapFeeder.TcPOU
(*
Nazwa:			P08_CapFeeder
Opis:			Stacja podajnika nasadek
Wersja:			v0.1
Data:			2022-07-13
Autor:			DJ,DP
Urzadzenia:		
Konfiguracja:	
Info:

*)
PROGRAM P08_CapFeeder
VAR_INPUT

END_VAR
VAR
	fbCapFeeder						: FB_CapFeeder;
	fbCapFeederState				: FB_State;	
	eCapFeederState					: E_Station;
	eCapFeederRunningState			: E_CapFeederState; 		// Stan pracy 
	
	IbCapFeederHeightEncoderSetCDone	AT %I*: BOOL;
	IudiCapFeederHeightEncoderCV        AT %I*: UDINT; 
	QbCapFeederHeightEncoderSetC 		AT %Q*: BOOL;		
	QudiCapFeederHeightEncoderSetCV     AT %Q*: UDINT; 	

	QbCapFeederHeightUpCmd 			AT %Q*: BOOL; 					// Wyjście sterujące podnośnikiem podajnika nakrętek, Silnik w górę
	QbCapFeederHeightDownCmd 		AT %Q*: BOOL; 				 	// Wyjście sterujące podnośnikiem podajnika nakrętek, Silnik w dół
	
	QbCapFeederSorterEngine			AT %Q*: BOOL; 					// Wyjście silnikiem sortera
	QbCapFeederSorterAir 			AT %Q*: BOOL; 					// Wyjście sterujące szybkim zaworem wydmuchu
	QbCapFeederSorterAir2 			AT %Q*: BOOL; 					// Wyjście sterujące szybkim zaworem wydmuchu
	
	IbCapFeederSorterCapSensor 		AT %I*: BOOL;					// Wejście z czujnika ultradzwiękowego nasadki sortera
	IbCapFeederFullSleeveSensor		AT %I*: BOOL;					// Wejście przepełnienia rękawa sortera
	IbCapFeederLevelSensor			AT %I*: BOOL;					// Wejście czujnika poziomu sortera

	
	IbFuseCapFeederEngineOK			AT %I*: BOOL;					//Bezpiecznik silnika sortera OK

	IbCapFeederHomingSensor			AT %I*: BOOL;					// Czujnnik bazowania, sorter w gornej pozycji 
	
	QnCapFeederSorterVelocitySV 	AT %Q*: UDINT; 		// Nastawa prędkości
	InCapFeederSorterVelocityCV 	AT %I*: UDINT;		
	InCapFeederSorterSTW 			AT %I*: UINT; 		// Statusword transportera wejściowo wyjściowego
	QnCapFeederSorterCTW 			AT %Q*: UINT;  		// Controlword transportera we/wy
	IbCapFeederSorterWcState		AT %I*: BOOL; 		// Statusword transportera wejściowo wyjściowego

	IbCapFeederPipeSensor			AT %I*: BOOL;		// Czujnik obecnośći flipflopa w rękawie
	
	TimerCapFeederEnable: TOF;
	rtEnable: R_TRIG;
	tonCapFeederEnable: TON;
	
	QbCapFeederGate1 			AT %Q*: BOOL; 					// Wyjście sterujące słabanem #1 w rękawe
	QbCapFeederGate2 			AT %Q*: BOOL; 					// Wyjście sterujące słabanem #1 w rękawe
	
	
	
	bTestW1: BOOL;
END_VAR

aCapFeeder();
aCapFeederWarnings();
QbCapFeederSorterAir2 :=	QbCapFeederSorterEngine OR QbCapFeederSorterAir; //Dodatkowy przedmuch

(* BAZOWANIE - ZMIAN*)
tonCapFeederEnable (IN:=fbCapFeeder.bEnable,PT:=T#5S); (*Dodany ton bo Wizka zjebnie wgrywa zmienne, najpierw włacza Enabla a potem dopiero wybiera recepture*)
rtEnable(CLK:=tonCapFeederEnable.Q,Q=>);
IF rtEnable.Q AND (P00_PackML.fbPMLAuto.ePMLState = E_PMLState.ePMLState_IDLE OR P00_PackML.fbPMLAuto.ePMLState = E_PMLState.ePMLState_EXECUTE)   THEN
		VIS.bCapFeederHeightSet:=TRUE;
ELSIF fbCapFeeder.eState=E_Station.eHomingDone  OR VIS.bErrorOccure THEN
 		VIS.bCapFeederHeightSet:=FALSE;
END_IF
(*KONIEC BAZOWANIE - ZMIANA*)

(*Opoznienie wyłączanie enabla*)
TimerCapFeederEnable(IN:=bCapFeederEnable, PT:=T#2S);

fbCapFeederState(
	eState:=eCapFeederState , 
	bRun:=VIS.bCapFeederRun,	
	eCapFeederRunningState:=eCapFeederRunningState , 
	sStateDesc=> VIS.sCapFeederState,
	iState=>VIS.iCapFeederState	);

ACTION aCapFeeder:
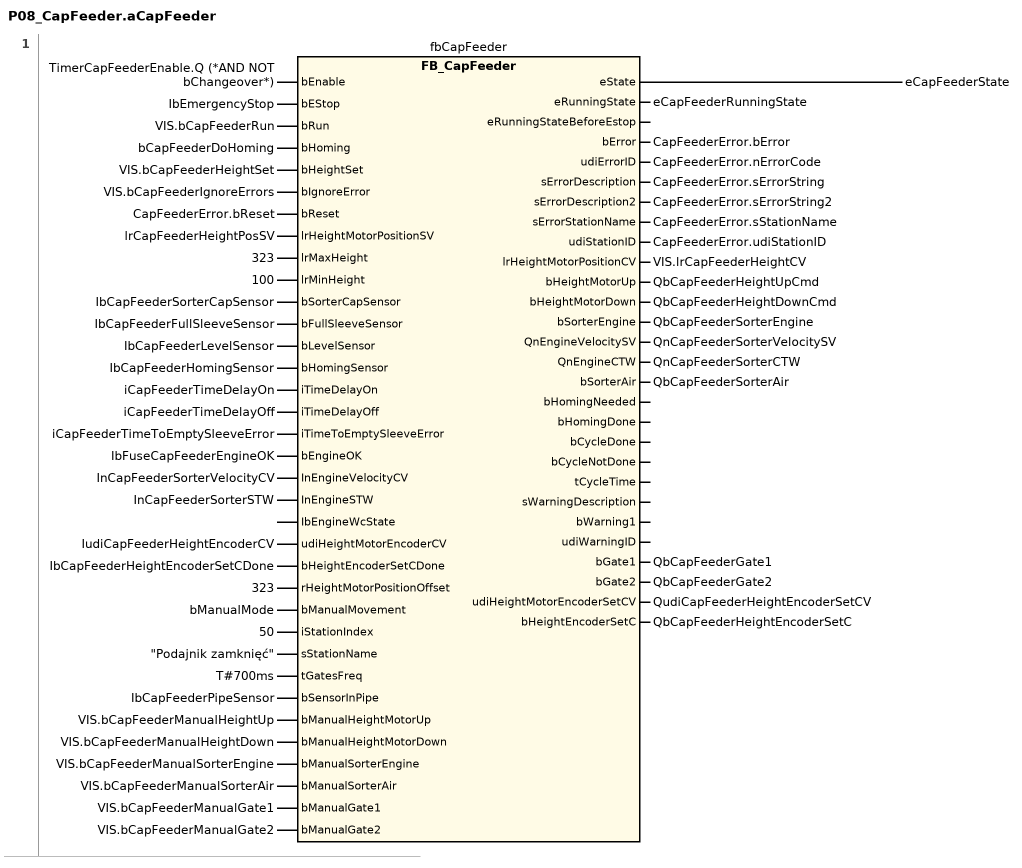
// NETWORK 1
fbCapFeeder(
    bEnable := TimerCapFeederEnable.Q (*AND NOT bChangeover*),
    bEStop := IbEmergencyStop,
    bRun := VIS.bCapFeederRun,
    bHoming := bCapFeederDoHoming,
    bHeightSet := VIS.bCapFeederHeightSet,
    bIgnoreError := VIS.bCapFeederIgnoreErrors,
    bReset := CapFeederError.bReset,
    lrHeightMotorPositionSV := lrCapFeederHeightPosSV,
    lrMaxHeight := 323,
    lrMinHeight := 100,
    bSorterCapSensor := IbCapFeederSorterCapSensor,
    bFullSleeveSensor := IbCapFeederFullSleeveSensor,
    bLevelSensor := IbCapFeederLevelSensor,
    bHomingSensor := IbCapFeederHomingSensor,
    iTimeDelayOn := iCapFeederTimeDelayOn,
    iTimeDelayOff := iCapFeederTimeDelayOff,
    iTimeToEmptySleeveError := iCapFeederTimeToEmptySleeveError,
    bEngineOK := IbFuseCapFeederEngineOK,
    InEngineVelocityCV := InCapFeederSorterVelocityCV,
    InEngineSTW := InCapFeederSorterSTW,
    udiHeightMotorEncoderCV := IudiCapFeederHeightEncoderCV,
    bHeightEncoderSetCDone := IbCapFeederHeightEncoderSetCDone,
    rHeightMotorPositionOffset := 323,
    bManualMovement := bManualMode,
    iStationIndex := 50,
    sStationName := "Podajnik zamknięć",
    tGatesFreq := T#700ms,
    bSensorInPipe := IbCapFeederPipeSensor,
    bManualHeightMotorUp := VIS.bCapFeederManualHeightUp,
    bManualHeightMotorDown := VIS.bCapFeederManualHeightDown,
    bManualSorterEngine := VIS.bCapFeederManualSorterEngine,
    bManualSorterAir := VIS.bCapFeederManualSorterAir,
    bManualGate1 := VIS.bCapFeederManualGate1,
    bManualGate2 := VIS.bCapFeederManualGate2,
    eRunningState => eCapFeederRunningState,
    bError => CapFeederError.bError,
    udiErrorID => CapFeederError.nErrorCode,
    sErrorDescription => CapFeederError.sErrorString,
    sErrorDescription2 => CapFeederError.sErrorString2,
    sErrorStationName => CapFeederError.sStationName,
    udiStationID => CapFeederError.udiStationID,
    lrHeightMotorPositionCV => VIS.lrCapFeederHeightCV,
    bHeightMotorUp => QbCapFeederHeightUpCmd,
    bHeightMotorDown => QbCapFeederHeightDownCmd,
    bSorterEngine => QbCapFeederSorterEngine,
    QnEngineVelocitySV => QnCapFeederSorterVelocitySV,
    QnEngineCTW => QnCapFeederSorterCTW,
    bSorterAir => QbCapFeederSorterAir,
    bGate1 => QbCapFeederGate1,
    bGate2 => QbCapFeederGate2,
    udiHeightMotorEncoderSetCV => QudiCapFeederHeightEncoderSetCV,
    bHeightEncoderSetC => QbCapFeederHeightEncoderSetC); // FB_CapFeeder
eCapFeederState := fbCapFeeder.eState;
END_ACTION

ACTION aCapFeederWarnings:
// Sorter nasadek

IF fbCapFeeder.bWarning1 AND NOT CapFeederWarning[0].bWarning THEN
	CapFeederWarning[0].bWarning										:= TRUE;
	CapFeederWarning[0].udiWarningCode									:= 33;	
	CapFeederWarning[0].sDescription									:= 'Podajnik nasadek | Niski poziom nasadek';
ELSIF NOT fbCapFeeder.bWarning1  AND CapFeederWarning[0].bAcknowledge THEN
	CapFeederWarning[0].bWarning										:= FALSE;
	CapFeederWarning[0].bAcknowledge									:= FALSE;
	VIS.uliWarningAcknowledge.14 										:= FALSE;
ELSIF CapFeederWarning[0].bAcknowledge THEN
	CapFeederWarning[0].bAcknowledge									:= TRUE;
END_IF
END_ACTION

END_PROGRAM

// ---- POUs/FB/FB_CapFeeder.TcPOU
(*
Nazwa:			FB_CapFeederV2
Opis:			Sorter nasadek i podajnik nasadek z podnośnikiem JIESANG
Wersja:			v0.1
Data:			2022-07-07
Autor:			DJA
Urzadzenia:		Silnik sortera, podnośnik JIESANG, Wydmuch, czujniki zapełnienia rękawa
Konfiguracja:	
Info:
-poprawiona wersja sortera względem poprzedniej, przerobione na aktualny standard State i RunningState
*)


FUNCTION_BLOCK FB_CapFeeder
VAR_INPUT
	
	bEnable						: BOOL;					//Zezowlenie na pracę stacji sprawdzania
	bEStop						: BOOL;					//Stop Awaryjny nieaktywny
	bRun						: BOOL;					//Włączenie sortera nasadek
	bHoming						: BOOL;					//Zezwolenie na wykonanie bazowania i pozycjonowania stacji sprawdzania
	bHeightSet					: BOOL;					// Bit do bazowania stacji na ustaloną wysokość 
	bIgnoreError				: BOOL;					//Ignorowania błędów cyklu pracy
	bReset						: BOOL;					//Reset błędu, jeśli w stanie "eError"
	lrHeightMotorPositionSV		: LREAL;				//Wysokość zadana na której ma znajdować się stacja
	lrMaxHeight					: LREAL;				//Maksymalna wysokość stacji sprawdzania
	lrMinHeight					: LREAL;				//Minimalna wysokość stacji sprawdzania
	bSorterCapSensor 			: BOOL;					// Wejście z czujnika ultradzwiękowego nasadki sortera
	bFullSleeveSensor			: BOOL;					// Wejście przepełnienia rękawa sortera
	bLevelSensor				: BOOL;					// Czujnik poziomu
	bHomingSensor				: BOOL;					// Wejscie czujnika bazowania napedu 
	iTimeDelayOn				: INT; 					//Czas na właczenie silnika sortera po zaniku sygnału przepełnienia z rękawa
	iTimeDelayOff				: INT; 					// Czas na wylączenie silnika sortera po wykryciu sygnału przepełnienia z rękawa sortera
	iTimeToEmptySleeveError		: INT;					// Czas do włączenia alrmu pustego rękawa
	bEngineOK					: BOOL;					//Wejście czujnika zabezpieczenia silnika 
	InEngineVelocityCV 			: UDINT;		
	InEngineSTW 				: UINT; 				// Statusword transportera wejściowo wyjściowego
	IbEngineWcState				: BOOL; 				// Statusword transportera wejściowo wyjściowego
	udiHeightMotorEncoderCV		: UDINT;
	bHeightEncoderSetCDone		: BOOL;	
	
	rHeightMotorPositionOffset 	: REAL;					//Wysokość bazowania podnośnika
	bManualMovement				: BOOL; 				//Uruchomienie trybu ruchów ręcznych
	iStationIndex				: UDINT;				// Indywidualny numer stacji
	sStationName				: WSTRING;				// Nazwa stacji
	
	tGatesFreq					:	TIME;
	
	bSensorInPipe				:	BOOL;				// Czujnik obecnośći flipflopa w rękawie
END_VAR

VAR_OUTPUT
	eState						: E_Station;			// Aktualny stan stacju
	eRunningState				: E_CapFeederState;		// Stan pracy stacji
	eRunningStateBeforeEstop	: E_CapFeederState;  	// Stan przed Estope
	bError						: BOOL;					// Błąd stacji
	udiErrorID					: UDINT;				// Nr blędu przeciągania formatek
	sErrorDescription			: STRING(200);			// Opis błędu
	sErrorDescription2			: STRING(200);			// Opis błędu
	sErrorStationName			: STRING;				// Nazwa stacj
	udiStationID				: UDINT;				// Nr stacj
	lrHeightMotorPositionCV		: LREAL;				//Aktualna pozycja podnośnika stacji
	bHeightMotorUp				: BOOL;					//Sterowanie silnikiem podnośnika  - RUCH W GÓRĘ
	bHeightMotorDown			: BOOL;					//Sterowanie silnikiem podnośnika  - RUCH W DÓŁ
	bSorterEngine 				: BOOL; 				// Sterowanie silnikiem sortera
	QnEngineVelocitySV 			: UDINT; 				// Nastawa prędkości
	QnEngineCTW 				: UINT;  				// Controlword transportera we/wy	
	bSorterAir 					: BOOL; 				// Sterowanie szybkim zaworem wydmuchu
	bHomingNeeded				: BOOL;					// Wymagane ponowne bazowanie (blad podczas bazowania lub stop awaryjny)
	bHomingDone					: BOOL;					// Stacja zbazowana 
	bCycleDone					: BOOL;					// Sygnał o zakończeniu cyklu
	bCycleNotDone				: BOOL;					// Sygnał o niezakończonym cyklu
	tCycleTime					: TIME;	 				// Czas cyklu 
	sWarningDescription			: STRING;
	bWarning1					: BOOL;
	udiWarningID				: UDINT;
	
	bGate1						:	BOOL;	//Szlaban w podajniku nakrętek #1
	bGate2						:	BOOL;	//Szlaban w podajniku nakrętek #2
	
	udiHeightMotorEncoderSetCV	: UDINT;		
	bHeightEncoderSetC			: BOOL;	
	
END_VAR

VAR_IN_OUT
	bManualHeightMotorUp		: BOOL;					//Ruch ręczny podnośnika stacji w górę
	bManualHeightMotorDown		: BOOL;					//Ruch ręczny podnośnika stacji w dół
	bManualSorterEngine			: BOOL;					//Ręczne włączenie silnika sortera
	bManualSorterAir			: BOOL;					//Ręczne włączenie zaworu wydmuchu
	
	bManualGate1				:	BOOL;									// Szlaban #1 w rękawe
	bManualGate2				:	BOOL;									// Szlaban #2 w rękawe		
	
END_VAR

VAR
	i							:	INT;
	aBufferedSensorValue		:	ARRAY[0..50] OF BOOL;	
	iValvesCycleCase			:	INT;
	rtOutSensor					:	R_TRIG;

	// State
	eLastState					: E_Station;			//Stan ogólny bloku
	eLastStateTemp				: E_Station;			//Stan ogólny bloku
	eLastRunningState			: E_CapFeederState;		//Stan podbloku
	eLastRunningStateTemp		: E_CapFeederState;		//Stan podbloku

	fbHeightMotorEncoder		: FB_JiesangActuatorEncoderModul;				// Blok enkodera podnośnika chwytaka stabilizującego pod zakręcarką	
	bHeightMotorEncoderCounterReset						:BOOL; 				// Sygnał resetu enkodera
	lrLastHeightMotorPositionCV		: LREAL;				// Pozycja podnośnika w poprzednim cyklu programu
	bHeightMotorEncoderHomed	: BOOL;					// Informacja od enkodera że jest zbazowany		
	bStateError					: BOOL;
	bManualPositionChanged		: BOOL;					// Ruszono Jiesanga w manualu => trzeba zdjąć bHomingDone

	tofHeightMotorDown			: TOF;					// Opóźnienie ruchu w dół, żeby nie przeciązać rozruchem układu
	rtEncoderHomed				: R_TRIG;				// Bit zakończenia enkodera
		
	tonHeightNoChange			: TON; 					// Timer wykrycia braku ruchu siłownika zmiany wysokości stacji
	tonHeightNoChangeTime		: TON; 					// Timer wykrycia braku ruchu siłownika zmiany wysokości stacji
	
	tonLimitPosMinReachedDelay	: TON;					// Timer osoiągniecia minimalnej wyskości 
	tonLimitPosMaxReachedDelay	: TON;					// Timer osiągnięcia maksymalnej wyskości
	tonSortingEngineOn			: TON;					// Opóźnienie po załączeniu napędu
	tonSortingEngineOff			: TON;					// Opóźnienie wyłączenia napędu
	tonSleeveFullEngineOn		: TON;					// Czas załączenia napędu po wykrciu braku nasadek
	tonEngineBlocked			: TON;					// Zablokowany silnik	
	rtCapSorterSensor			: R_TRIG;				// Triger
	tonTryUnblockWheel			: TON;					// Czas ruchu falownika w drugą stronę
	tofCapFeederSorterCapSensor	: TOF;					// Opóźnienie sygnału z czujnika obecności nasadki ultradzwiek
	tonCapFeederSorterCapSensor	: TON;					// Opóźnienie sygnału z czujnika obecności nasadki ultradźwięk
	tonAirBeforeStart			: TON;					// Czasówka opóźeniani przedmuchu
	tonAirBeforeStart2			: TON;					// Czasówka opóźeniani przedmuchu
	tonAirAfterStop				: TON;					// Czasówka przedmuchu po zatrzymaniu
	tonStoppingTime				: TON;					// Czasówka zbyt długiego zatrzymawania

	
	tonErrorHeightChange		: TON; 					// Timer błędu zacięcia się podnośnika
	tonEmptySleeveError			: TON;					// Timer pustego rękawa
	tonMaxHeightError			: TON;					// Timer ustawienia zbyt dużej wysokości stacji
	tonMinHeightError			: TON;					// Timer ustawienia zbyt małej wysokości stacji
	tonCycleTimer				: TON;					// Czasówka cyklu
	rtrigCycleTimerRead			: R_TRIG;				// Trigger do statystyk cyklu 
	
	tonSorterEngineError: TON;
	tonHomingSensor: TON;
	TimerOn: TON;
	TimerOff: TON;
	bImpOn: BOOL;
	rtCapFeederSorterCapSensor: R_TRIG;
	bBlowDelay: BOOL;
	tonbBlowDelay: TON;
	
	fbInverter: FB_MitsubishiInverter;
	tonInverterError: TON;
	(*Ostrzeżenia*)
	fbbLevelSensor:	FB_InputFilter;
	(*Inne*)	

	tonGates1	:	TON;	//Czasówka dla szlabanów w rękawe
	tonGates2	:	TON;	//Czasówka dla szlabanów w rękawe
	tonGates3	:	TON;	//Czasówka dla szlabanów w rękawe
	tonGates4	:	TON;	//Czasówka dla szlabanów w rękawe

		
	bGates	    :	BOOL;	//Controla szłabanow w rękawe  
	bTryUnblockWheel : BOOL;
	iTryUnblockWheel : INT;
	
	//Zmienne od EVENTLOGGER
	bAlarmInit 						: BOOL := TRUE; 
	nAlarmNumerator					: INT;
	arfbAlarm						: ARRAY[0..19] OF  FB_TcAlarm;		//Tablica bloczków błędów
	fbSourceInfo 					: FB_TcSourceInfo;
	iSourceInfo						: I_TcSourceInfo;
	sAlarmTest						: STRING;
	//Koniec zmiennych od EVENTLOGGER
END_VAR

//Wywołanie bloczków od stacji. Ważna jest ich kolejność!!!
ACT_Limits();
ACT_HeightMotor();
ACT_ErrorHandling();

ACT_Signals();
ACT_Control();
ACT_Inverter();
ACT_Statistic();
ACT_Status();
ACT_Warnings();
aStationID();	

lrLastHeightMotorPositionCV:=lrHeightMotorPositionCV;

ACTION ACT_Control:
	(*****Wyłączenie enable*****)
	IF NOT bEnable THEN
		IF eState <> E_Station.eDisabled AND eState <> E_Station.ePreparingToDisable THEN
				eState 				:= E_Station.ePreparingToDisable; 
		END_IF	
	END_IF

	(*****Estop*****)
	IF NOT bEstop  THEN	
		IF eState <> E_Station.eAborted AND eState <> E_Station.eAborting AND eState <> E_Station.eDisabled THEN
				eState 				:= E_Station.eAborting; 
		END_IF
	END_IF


	CASE eState OF
//--------------------------------------------------------------------------------
// Stan maszyny po wyłączeniu i przygotowanie do uruchomienia
	E_Station.eDisabled: 					// Stan nieaktywnosci (Stacja wyłączona) 
	
		IF bEnable THEN
			eState 				:= E_Station.ePreparingToReady; 
		END_IF 
		
//--------------------------------------------------------------------------------
// Stan maszyny po zatrzymaniu awaryjnym   
	E_Station.eAborted: 					// Stan bezpiecznego zatrzymania (po Abortingu) 

		IF bEStop THEN
			eState 				:= E_Station.ePreparingToReady;
		END_IF
		
//--------------------------------------------------------------------------------
// Stan maszyny naciśnieciu estopa 	
	E_Station.eAborting:                 	// Stan bezpiecznego zatrzymywania (po EStopie)
		bGate1:= FALSE;
		bGate2:= FALSE;
	
		ACT_ResetCommands();

		eState 						:=  E_Station.eAborted;  
		eRunningState				:=	E_CapFeederState.eReady;
		
//--------------------------------------------------------------------------------
// Stan masyzny po wykryciu błędu			
	E_Station.eError:                 	 	// Stan błędu 	
		
		ACT_ResetCommands();
		
		IF bReset THEN
			eState 				:= E_Station.eResetting;
			bError := FALSE;
		END_IF
		
//--------------------------------------------------------------------------------
// Stan masyzny po wykryciu błędu
	E_Station.eResetting:					// Stan resetowania bledu (po Errorze)
// 			CASE udiErrorID-udiStationIndex OF
// 		
// 				//Error 8 - Błąd falownika
// 				9:
// 					fbInverter.bReset	:= TRUE;
// 					bError 				:= FALSE;
// 				ELSE
// 					bError := FALSE;	
// 			END_CASE		
		
		IF NOT bError AND fbInverter.eState = E_Station.eReady THEN
			fbInverter.bReset	:= FALSE;	
			{warning 'Sprawdzić błąd falownika CapFeeder'}
			udiErrorID 			:=	0;
			sErrorDescription 	:=	'';
			eState 				:=	E_Station.ePreparingToReady;
			eRunningState		:=	E_CapFeederState.eReady;
		ELSE
			eState 				:=	E_Station.eError;
		END_IF
    
//--------------------------------------------------------------------------------
// Stan ruchoow manualnych
	E_Station.eManualMovement:     			// Stan ruchów manualnych  
   
		ACT_ManualMovements();
		IF bManualHeightMotorUp OR bManualHeightMotorDown THEN
				bManualPositionChanged		:= TRUE;
			END_IF
		//Wyjście z trybu serwisowego
		IF NOT bManualMovement THEN
			
			bHeightMotorUp				:=	FALSE;
			bHeightMotorDown			:=	FALSE;
			IF bManualPositionChanged THEN
				bHomingDone				:= FALSE;
				bManualPositionChanged	:= FALSE;
			END_IF
			
			eState:=E_Station.eReady;
		END_IF
		

//--------------------------------------------------------------------------------
// Stan rozpoczecia bazowania
	E_Station.eHoming:						// Stan bazowania 
		
		ACT_Homing();
		IF NOT bHoming AND NOT bHeightSet THEN
			bHeightMotorDown					:=	FALSE;
			bHeightMotorUp						:=	FALSE;
		   eState								:=E_Station.ePreparingToReady;
		END_IF		
		
//--------------------------------------------------------------------------------
// Stan zakończenia bazowania
	E_Station.eHomingDone:                  // Stan wykonania bazowania 
	
		bHeightMotorDown					:=	FALSE;
		bHeightMotorUp						:=	FALSE;
		bHeightMotorEncoderCounterReset		:=	FALSE;
		bHomingDone							:=	TRUE;
		IF NOT bHoming AND NOT bHeightSet THEN
		   eState:=E_Station.eReady;
		END_IF
		
//--------------------------------------------------------------------------------
// Stan przygotowania do gotowości
	E_Station.ePreparingToReady:            // Stan przygotowywania do gotowosci (zawsze przed Ready)  
		
		bGate1:= FALSE;
		bGate2:= FALSE;
	
		bSorterEngine:=FALSE;
		bSorterAir:=FALSE;
		
		eRunningState:=E_CapFeederState.eReady;
		eState:=E_Station.eReady;	
		
//-------------------------------------------------------------------------------
// Stan przygotowania do wyłączenia maszyny
	E_Station.ePreparingToDisable:          // Stan przygotowywania do nieaktywnosci (po wyłączeniu Enable) 
		
		bGate1:= FALSE;
		bGate2:= FALSE;
	
		bSorterEngine:=FALSE;
		bSorterAir:=FALSE;
		bHeightMotorUp:= NOT tonHomingSensor.Q;
		bHeightMotorDown:=FALSE;	
		IF tonHeightNoChange.Q OR tonHeightNoChangeTime.Q THEN
			bHeightMotorUp			:=	FALSE;
			bHeightMotorDown		:=	FALSE;	
			eRunningState			:=	E_CapFeederState.eReady;		
			eState					:=	E_Station.eDisabled;
		END_IF	
			
//--------------------------------------------------------------------------------
// Stan gotowości
	E_Station.eReady:						// Stan gotowosci 
	
		IF bRun AND NOT bCycleDone AND NOT bCycleNotDone THEN
			eState 				:= E_Station.eStarting; 
		END_IF
		IF bHoming OR bHeightSet THEN
			bHomingDone							:=	FALSE;
			eState 								:= E_Station.eHoming; 
		END_IF
		IF bManualMovement THEN
			//Jeśli przejście w tryb ruchów manualnych przepisz wszystkie stany siłowników sterowanych przez moduł
			//aby zapobiec ewentualnym kolizjom po wejściu w tryb serwisowy
			
			bManualHeightMotorUp		:= bHeightMotorUp;
			bManualHeightMotorDown		:= bHeightMotorDown;
			bManualPositionChanged		:= FALSE;
			
			eState 						:= E_Station.eManualMovement; 
		END_IF
		IF NOT bRun THEN
			bCycleDone 			:= FALSE;
			bCycleNotDone 		:= FALSE;			
		END_IF
		
//--------------------------------------------------------------------------------
// Stan zatrzymywania
	E_Station.eStopping:					// Stan zatrzymywania 
		
		bSorterAir 		:= 	TRUE;
		bSorterEngine 	:=	FALSE;
		IF tonStoppingTime.Q THEN
			ACT_ResetCommands();
			eRunningState							:= E_CapFeederState.eReady;
			eState									:= E_Station.eReady;
		END_IF

		
//--------------------------------------------------------------------------------
// Stan uruchomienia lini ( po eReady)
	E_Station.eStarting:                  	// Stan uruchamiania (po Ready)
		iValvesCycleCase		:=0;
		eState					 := E_Station.eRunning; 

//--------------------------------------------------------------------------------
// Stan wykonywania pracy
	E_Station.eRunning:               		// Stan wykonywania cyklu (po Startingu), w tym stanie osobny

		ACT_Running();
		IF NOT bRun THEN 					(*Przerywanie cyklu*)
			eState				:= E_Station.eStopping;
			//bCycleNotDone		:= TRUE;
		END_IF
		(*IF bCycleDone OR bCycleNotDone THEN (*Cykl zakończony*)
			eState 				 := E_Station.eReady;
		END_IF*)						
		
		
END_CASE
END_ACTION

ACTION ACT_ErrorHandling:
// Alarm_0400	400	Error	Blokada podnośnika lub brak zasilania - sprawdź czujnik lub odblokuj mechanicznie
// Alarm_0401	401	Error	Bład zabezpieczenia silnika - sprawdź wyłącznik
// Alarm_0402	402	Error	Pusty rękaw sortera - uzupełnij nasadki
// Alarm_0403	403	Error	Wartość zadana wysokości jest większa od maksymalnej - zmień ustawienia w recepturze {0}
// Alarm_0404	404	Error	Wartość zadana wysokości jest mniejsza od minimalnej - zmień ustawienia w recepturze {0}
// Alarm_0405	405	Error	Błąd falownika

IF bAlarmInit THEN
    bAlarmInit := FALSE; 
	fbSourceInfo.Clear();
	fbSourceInfo.sName:=wsLiteral_TO_UTF8(sStationName);//'Machine';
	fbSourceInfo.nId:=udiStationID;//2700;
	// Alarm_0400	400	Error	Blokada podnośnika lub brak zasilania - sprawdź czujnik lub odblokuj mechanicznie
    arfbAlarm[0].CreateEx(stEventEntry := TC_EVENTS.AlarmClass.Alarm_0400, bWithConfirmation:= FALSE,  ipSourceInfo:= fbSourceInfo); 
	// Alarm_0401	401	Error	Bład zabezpieczenia silnika - sprawdź wyłącznik
	arfbAlarm[1].CreateEx(stEventEntry := TC_EVENTS.AlarmClass.Alarm_0401, bWithConfirmation:= FALSE,  ipSourceInfo:= fbSourceInfo);
	// Alarm_0402	402	Error	Pusty rękaw sortera - uzupełnij nasadki
	arfbAlarm[2].CreateEx(stEventEntry := TC_EVENTS.AlarmClass.Alarm_0402, bWithConfirmation:= FALSE,  ipSourceInfo:= fbSourceInfo);
	// Alarm_0403	403	Error	Wartość zadana wysokości jest większa od maksymalnej - zmień ustawienia w recepturze {0}
	arfbAlarm[3].CreateEx(stEventEntry := TC_EVENTS.AlarmClass.Alarm_0403, bWithConfirmation:= FALSE,  ipSourceInfo:= fbSourceInfo);
	// Alarm_0404	404	Error	Wartość zadana wysokości jest mniejsza od minimalnej - zmień ustawienia w recepturze {0}
	arfbAlarm[4].CreateEx(stEventEntry := TC_EVENTS.AlarmClass.Alarm_0404, bWithConfirmation:= FALSE,  ipSourceInfo:= fbSourceInfo);
	// Alarm_0405	405	Error	Błąd falownika
	arfbAlarm[5].CreateEx(stEventEntry := TC_EVENTS.AlarmClass.Alarm_0405, bWithConfirmation:= FALSE,  ipSourceInfo:= fbSourceInfo);
END_IF




//OBSŁUGA BŁĘDÓW STACJI SPRAWDZANIA
//************LISTA BŁĘDÓW***************
bStateError:= (eState=E_Station.eError) OR (eState=E_Station.eResetting) OR bIgnoreError;

//************LISTA BŁĘDÓW***************

//Error 1 - podnośnik nie porusza się pomimo wysterowania 
tonErrorHeightChange(IN:=(bHeightMotorUp OR bHeightMotorDown) AND lrLastHeightMotorPositionCV=lrHeightMotorPositionCV, PT:=T#3S);
tonEmptySleeveError(IN:=NOT bFullSleeveSensor AND bRun, PT:=INT_TO_TIME(iTimeToEmptySleeveError)*1000); //Było 30, teraz jest z receptur
tonMaxHeightError(IN:=lrHeightMotorPositionSV>lrMaxHeight AND NOT bHomingNeeded AND eState=E_Station.eReady,PT:=T#30S);
tonMinHeightError(IN:=lrHeightMotorPositionSV<lrMinHeight AND NOT bHomingNeeded AND eState=E_Station.eReady,PT:=T#30S);
tonSorterEngineError(IN:= NOT bEngineOK AND bSorterEngine, PT:=T#3S);
tonInverterError(IN:=fbInverter.bError AND NOT bStateError, PT:=T#3S);

IF (bEnable OR (eState = E_Station.ePreparingToDisable)) AND NOT bIgnoreError THEN
	// Alarm_0400	400	Error	Blokada podnośnika lub brak zasilania - sprawdź czujnik lub odblokuj mechanicznie
	IF tonErrorHeightChange.Q THEN
		IF NOT arfbAlarm[0].bActive THEN
			arfbAlarm[0].Raise(nTimeStamp:=0);
		END_IF
	ELSE	
		IF  arfbAlarm[0].bActive AND bReset THEN
			arfbAlarm[0].Clear(nTimeStamp:=0, bResetConfirmation:= FALSE);
		END_IF
// 		bError:=TRUE;
// 		udiErrorID:=1;
// 		udiErrorID:= udiErrorID+udiStationIndex;
// 		sErrorDescription:='Blokada podnośnika lub brak zasilania - sprawdź czujnik lub odblokuj mechanicznie';	
// 		sErrorDescription2:='';
	END_IF
	
	// Alarm_0401	401	Error	Bład zabezpieczenia silnika - sprawdź wyłącznik
	IF tonSorterEngineError.Q THEN
		IF NOT arfbAlarm[1].bActive THEN
			arfbAlarm[1].Raise(nTimeStamp:=0);
		END_IF
	ELSE	
		IF  arfbAlarm[1].bActive AND bReset THEN
			arfbAlarm[1].Clear(nTimeStamp:=0, bResetConfirmation:= FALSE);
		END_IF
// 		bError:=TRUE;
// 		udiErrorID:=2;
// 		udiErrorID:= udiErrorID+udiStationIndex;
// 		sErrorDescription:='Bład zabezpieczenia silnika - sprawdź wyłącznik';	
// 		sErrorDescription2:='';	
	END_IF
	// Alarm_0402	402	Error	Pusty rękaw sortera - uzupełnij nasadki
	//Error 3 - Pusty rekaw sortera nasadek
	IF tonEmptySleeveError.Q THEN
		IF NOT arfbAlarm[2].bActive THEN
			arfbAlarm[2].Raise(nTimeStamp:=0);
		END_IF
	ELSE	
		IF  arfbAlarm[2].bActive AND bReset THEN
			arfbAlarm[2].Clear(nTimeStamp:=0, bResetConfirmation:= FALSE);
		END_IF
// 		bError:=TRUE;
// 		udiErrorID:=3;
// 		udiErrorID:= udiErrorID+udiStationIndex;
// 		sErrorDescription:='Pusty rękaw sortera - uzupełnij nasadki';
// 		sErrorDescription2:='';
	END_IF
	
